# B&R Automation Studio project PLC code - cp (part 24)

```c
		case 8:
			strcpy(txStateDesc, "Waiting homing ");
			TEST_BUSY_CONDITION( !gBlock[1].Status.Motor.xBarsHomed );
			nextState();
			break;

		case 9:

			iTestState = 0;
			TEST_DONE;

			break;

		default:
			break;
	}

}

_TEST test_RemoveTrayMovementMemoryWithKey(void)
{ // Related to https://jira.efi.com/browse/CUBE-963

	if (!gSafetyController.Parameters.xInstalled ){
		iTestState = 0;

		//This 2 lines just for the last TestCase
		strcpy(txTest, "BlockTests Finished!! Congrats!");
		strcpy(txStateDesc, "--");

		TEST_DONE;
	}

	strcpy(txTest, "test_RemoveTrayMovementMemoryWithKey");
	if (strcmp(&txTest, &gSimMachine.Commands.LogTests.Text) != 0){
		strcpy(gSimMachine.Commands.LogTests.Text, txTest); gSimMachine.Commands.LogTests.xCommand = TRUE;
	}
	switch (iTestState)
	{
		case 0:
			gSimMachine.Commands.xToZero = TRUE;
			nextState();
			break;

		case 1:
			strcpy(txStateDesc, "Going to Zero");
			TEST_BUSY_CONDITION( !gMachine.St.Mode.xZero );
			nextState();
			break;

		case 2:
			gSimMachine.Commands.xToAuto = TRUE;
			strcpy(txStateDesc, "Going to Auto");
			TEST_BUSY_CONDITION( !gMachine.St.Mode.xAuto );
			nextState();
			break;

		case 3:
			strcpy(txStateDesc, "Going to Cap");
			TEST_BUSY_CONDITION( gMachine.St.exec.slow < exTimesPreSlow + 3 ); //We'll wait xx scan cycles
			TEST_BUSY_CONDITION( !gMachine.St.Position.xInCap );
			nextState();
			break;

		case 4:
			gSimMachine.Commands.xToZero = TRUE;
			nextState();
			break;

		case 5:
			strcpy(txStateDesc, "Going to Zero");
			TEST_BUSY_CONDITION( !gMachine.St.Mode.xZero );
			nextState();
			break;

		case 6:
			gSimMachine.Commands.xToManual = TRUE;
			strcpy(txStateDesc, "Going to Manual");
			TEST_BUSY_CONDITION( !gMachine.St.Mode.xManual );
			nextState();
			break;

		case 7:
			strcpy(txStateDesc, "Activating the Key");
			TEST_BUSY_CONDITION( gMachine.St.exec.slow < exTimesPreSlow + 2 ); //We'll wait xx scan cycles
			gSimSafetyController.Inputs.xPrinterMaintenanceKey = TRUE;
			nextState();
			break;

		case 8:
			strcpy(txStateDesc, "Send the order to move tray out");
			TEST_BUSY_CONDITION( gMachine.St.exec.slow < exTimesPreSlow + 5 ); //We'll wait xx scan cycles
			gBlock[1].commands.Manual.xManTrayOut = TRUE;
			nextState();
			break;

		case 9:
			strcpy(txStateDesc, "Checking NOT movement");
			TEST_BUSY_CONDITION( gMachine.St.exec.slow < exTimesPreSlow + 20 ); //We'll wait xx scan cycles
			TEST_ASSERT( gBlock[1].In.xTrayIn );
			nextState();
			break;

		case 10:
			strcpy(txStateDesc, "Remove Key");
			TEST_BUSY_CONDITION( gMachine.St.exec.slow < exTimesPreSlow + 5 ); //We'll wait xx scan cycles
			gSimSafetyController.Inputs.xPrinterMaintenanceKey = FALSE;
			nextState();
			break;

		case 11:
			strcpy(txStateDesc, "Checking NOT movement");
			TEST_BUSY_CONDITION( gMachine.St.exec.slow < exTimesPreSlow + 20 ); //We'll wait xx scan cycles
			TEST_ASSERT( gBlock[1].In.xTrayIn );
			nextState();
			break;

		case 12:

			iTestState = 0;

			//This 2 lines just for the last TestCase
			strcpy(txTest, "BlockTests Finished!! Congrats!");
			strcpy(txStateDesc, "--");

			TEST_DONE;
			break;

		default:
			break;
	}

}

/*
B+R UnitTest: This is generated code.
Do not edit! Do not move!
Description: UnitTest Testprogramm infrastructure (TestSet).
LastUpdated: 2024-03-01 15:54:59Z
By B+R UnitTest Helper Version: 2.0.1.59
*/
UNITTEST_FIXTURES(fixtures)
{
	new_TestFixture("test_CleanMachine", test_CleanMachine),
	new_TestFixture("test_GoDownWithTrayError", test_GoDownWithTrayError),
	new_TestFixture("test_GoUpWithTrayError", test_GoUpWithTrayError),
	new_TestFixture("test_GoToPrintInLaboratory", test_GoToPrintInLaboratory),
	new_TestFixture("test_GoToPrintInProduction", test_GoToPrintInProduction),
	new_TestFixture("test_TraySensorErrorWhilePrinting", test_TraySensorErrorWhilePrinting),
	new_TestFixture("test_GoToPrintWhileNSensorsCalibrationAreBeingChecked", test_GoToPrintWhileNSensorsCalibrationAreBeingChecked),
	new_TestFixture("test_ToNotChangeBarsPositionSetpointWhileDetectionSystemMotorIsBeingPositioned", test_ToNotChangeBarsPositionSetpointWhileDetectionSystemMotorIsBeingPositioned),
	new_TestFixture("test_GoToCleanBk1InLaboratory", test_GoToCleanBk1InLaboratory),
	new_TestFixture("test_ReturnToPrintFromClean", test_ReturnToPrintFromClean),
	new_TestFixture("test_RaiseBlocksToCapFromPrinting", test_RaiseBlocksToCapFromPrinting),
	new_TestFixture("test_StopWhenPrint_ReturnPrintingBeforCapPosition", test_StopWhenPrint_ReturnPrintingBeforCapPosition),
	new_TestFixture("test_CriticalAlarmWhilePrinting", test_CriticalAlarmWhilePrinting),
	new_TestFixture("test_GoToMaintenanceWhenInPrintingPositionAndCheckBarsNotMove", test_GoToMaintenanceWhenInPrintingPositionAndCheckBarsNotMove),
	new_TestFixture("test_CuringLedBarJamAlarm", test_CuringLedBarJamAlarm),
	new_TestFixture("test_CameraJamAlarm", test_CameraJamAlarm),
	new_TestFixture("test_TrayBlockMaintenanceKey", test_TrayBlockMaintenanceKey),
	new_TestFixture("test_ToNotExecuteHomingBlockWhileMaintenanceKeyIsActivated", test_ToNotExecuteHomingBlockWhileMaintenanceKeyIsActivated),
	new_TestFixture("test_ToNotExecuteHomingIclaWhileMaintenanceKeyIsActivated", test_ToNotExecuteHomingIclaWhileMaintenanceKeyIsActivated),
	new_TestFixture("test_InkBarJamAlarm", test_InkBarJamAlarm),
	new_TestFixture("test_ToCleanTest", test_ToCleanTest),
	new_TestFixture("test_ToPrintPosTest", test_ToPrintPosTest),
	new_TestFixture("test_InksFailNotEnabledToPrint", test_InksFailNotEnabledToPrint),
	new_TestFixture("test_InksFailEnabledToPrint", test_InksFailEnabledToPrint),
	new_TestFixture("test_NoBentAlarmThcChgOTFly", test_NoBentAlarmThcChgOTFly),
	new_TestFixture("test_NoStopCleanWithNitrLow", test_NoStopCleanWithNitrLow),
	new_TestFixture("test_NoFeederBarsPos", test_NoFeederBarsPos),
	new_TestFixture("test_PneuBlockAls", test_PneuBlockAls),
	new_TestFixture("test_Noz2Jam", test_Noz2Jam),
	new_TestFixture("test_InkTanksAl", test_InkTanksAl),
	new_TestFixture("test_MaintenanceModeInk", test_MaintenanceModeInk),
	new_TestFixture("test_ChillerInksAl", test_ChillerInksAl),
	new_TestFixture("test_NotBlockInAutoIfNotHomed", test_NotBlockInAutoIfNotHomed),
	new_TestFixture("test_RemoveTrayMovementMemoryWithKey", test_RemoveTrayMovementMemoryWithKey),
};

UNITTEST_CALLER_COMPLETE_EXPLICIT(BlockTests, "BlockTests", 0, 0, fixtures, 0, 0, 0);
```

### Program Logical/UnitTest/Tests/CleaningTests

#### CleaningTests.var
```iecst
(********************************************************************
 * COPYRIGHT -- Bernecker + Rainer
 ********************************************************************
 * Program: CleaningTests
 * Author: Jorge Murria
 ********************************************************************
 * Local variables of program CleaningTests
 * General variables - do not change
 ********************************************************************)
(*Describe the test*)
VAR
	Testsuite : UtMgrTestSuite := (Name:='CleaningTests',Description:='Description of the Tests',Type:=utMgrTEST_TYPE_C,MetaInformation:='Some Meta Information can be added here');
END_VAR
(*Variables used in the tests*)
```

#### autoGeneratedFile.c
```c
/*
B+R UnitTest: This is generated code.
Do not edit! Do not move!
Description: UnitTest Testprogramm infrastructure (List of TestSets).
LastUpdated: 2020-05-18 14:29:28Z
By B+R UnitTest Helper Version: 2.0.1.59
*/
#include "UnitTest.h"

UNITTEST_TESTSET_DECLARATION  CleaningTests;

UNITTEST_TESTSET_FIXTURES(utTestSets)
{
	new_TestSet(CleaningTests),
};
UNTITTEST_TESTSET_HANDLER();
```

### Program Logical/UnitTest/Tests/ConsentTests (ANSIC)

#### ConsentTests.var - PVs for the program and test suite
```iecst
(********************************************************************
 * COPYRIGHT -- Bernecker + Rainer
 ********************************************************************
 * Program: ConsentTests
 * Author: Jorge Murria
 ********************************************************************
 * Local variables of program ConsentTests
 * General variables - do not change
 ********************************************************************)
(*Describe the test*)
VAR
	Testsuite : UtMgrTestSuite := (Name:='ConsentTests',Description:='Tests related to the Consents',Type:=utMgrTEST_TYPE_C,MetaInformation:='Some Meta Information can be added here');
END_VAR
(*Variables used in the tests*)
```

#### autoGeneratedFile.c - Auto generated code
```c
/*
B+R UnitTest: This is generated code.
Do not edit! Do not move!
Description: UnitTest Testprogramm infrastructure (List of TestSets).
LastUpdated: 2020-05-18 14:29:28Z
By B+R UnitTest Helper Version: 2.0.1.59
*/
#include "UnitTest.h"

UNITTEST_TESTSET_DECLARATION  ConsentTests;

UNITTEST_TESTSET_FIXTURES(utTestSets)
{
	new_TestSet(ConsentTests),
};
UNTITTEST_TESTSET_HANDLER();
```

### Program Logical/UnitTest/Tests/Cube (ANSIC)

#### Cube.var - PVs for the program and test suite
```iecst
(********************************************************************
 * COPYRIGHT -- Bernecker + Rainer
 ********************************************************************
 * Program: Cube
 * Author: Jorge Murria
 ********************************************************************
 * Local variables of program Cube
 * General variables - do not change
 ********************************************************************)
(*Describe the test*)
VAR
	Testsuite : UtMgrTestSuite := (Name:='Cube',Description:='Description of the Tests',Type:=utMgrTEST_TYPE_C,MetaInformation:='Some Meta Information can be added here');
END_VAR
(*Variables used in the tests*)
```

### Program Logical/UnitTest/Tests/FunctionsTests (ANSIC)

#### FunctionsTests.var - PVs for the program and test suite
```iecst
(********************************************************************
 * COPYRIGHT -- Bernecker + Rainer
 ********************************************************************
 * Program: FunctionsTests
 * Author: Jorge Murria
 ********************************************************************
 * Local variables of program FunctionsTests
 * General variables - do not change
 ********************************************************************)
(*Describe the test*)
VAR
	Testsuite : UtMgrTestSuite := (Name:='FunctionsTests',Description:='Description of the Tests',Type:=utMgrTEST_TYPE_C,MetaInformation:='Some Meta Information can be added here');
END_VAR
(*Variables used in the tests*)
VAR
	TestMediaTracking : ARRAY[0..iMAXTRACKINGARRAY] OF USINT; (*Matrix with the information about if there is Media in the position. Each position corresponds to a cm. Bit 0: L1 , Bit 1 L2*)
	TestBoolMediaTracking : ARRAY[0..iMAXTRACKINGARRAY] OF BOOL; (*Matrix with the information about if there is Media in the position. Each position corresponds to a cm. Bit 0: L1 , Bit 1 L2*)
	xTestMediaDetectionValuesL1 : ARRAY[0..THICK_MAX_UPDATE_VALUES] OF BOOL; (*Matrix with the information about if there is Media in the position. Each position corresponds to a cm. Bit 0: L1 , Bit 1 L2*)
	iIndexArray : UINT;
	TestMediaTrackingInside : ARRAY[0..THICK_MEDIATRACKING_MAX_MEDIA] OF stThicknessCtrl_MediaPosStatus; (*FIFO. Elements enter at the end, and go to First while exiting elements*)
	MediaConfigReseted : stThicknessCtrl_MediaConfig;
	IntensityOutput : ARRAY[0..THICKENERGY_MAX_LAMPS] OF INT;
	EnergyData : stThickCtrl_Energy;
	iIndexProcess : UINT;
	iIndexCross : UINT;
	udResult : UDINT;
	MediaData : stThicknessCtrl_MediaConfig;
	NewMediaStack : ARRAY[0..THICK_MEDIATRACKING_MAX_MEDIA] OF stThicknessCtrl_MediaPosStatus; (*FIFO Stack. Elements enter at the end, and go to First while exiting elements*)
	MediaEnergyRack : ARRAY[0..THICK_MEDIATRACKING_MAX_MEDIA_x2] OF stThickCtrl_Energy; (*Need the memory area for NewMedia and for MediaInside with full data*)
	Stack_iTotalNewMedia : UINT;
	Stack_iTotalNewMediaPos : UINT;
	EnergyRack_iIndex : USINT; (*Index of the next free rack in array*)
	Adresses : ARRAY[0..9] OF UDINT;
END_VAR
```

#### autoGeneratedFile.c - Auto generated code
```c
/*
B+R UnitTest: This is generated code.
Do not edit! Do not move!
Description: UnitTest Testprogramm infrastructure (List of TestSets).
LastUpdated: 2020-05-18 14:29:28Z
By B+R UnitTest Helper Version: 2.0.1.59
*/
#include "UnitTest.h"

UNITTEST_TESTSET_DECLARATION  FunctionsTests;

UNITTEST_TESTSET_FIXTURES(utTestSets)
{
	new_TestSet(FunctionsTests),
};
UNTITTEST_TESTSET_HANDLER();
```

### Program Logical/UnitTest/Tests/LineTests

#### LineTests.var
```iecst
(********************************************************************
 * COPYRIGHT -- Bernecker + Rainer
 ********************************************************************
 * Program: LineTests
 * Author: Jorge Murria
 ********************************************************************
 * Local variables of program LineTests
 * General variables - do not change
 ********************************************************************)
(*Describe the test*)
VAR
	Testsuite : UtMgrTestSuite := (Name:='LineTests',Description:='Description of the Tests',Type:=utMgrTEST_TYPE_C,MetaInformation:='Some Meta Information can be added here');
END_VAR
(*Variables used in the tests*)
```

#### autoGeneratedFile.c
```c
/*
B+R UnitTest: This is generated code.
Do not edit! Do not move!
Description: UnitTest Testprogramm infrastructure (List of TestSets).
LastUpdated: 2020-05-18 14:29:28Z
By B+R UnitTest Helper Version: 2.0.1.59
*/
#include "UnitTest.h"

UNITTEST_TESTSET_DECLARATION  LineTests;

UNITTEST_TESTSET_FIXTURES(utTestSets)
{
	new_TestSet(LineTests),
};
UNTITTEST_TESTSET_HANDLER();
```

#### LineTests.c
```c
/********************************************************************
 * COPYRIGHT -- Bernecker + Rainer
 ********************************************************************
 * Program: ConsentsTests
 * Author: Jorge Murria
 ********************************************************************
 * Prepare machine with basic test to allow proper behabior
 * and starting tasks
 ********************************************************************/

#include <bur/plctypes.h>

#ifdef _DEFAULT_INCLUDES
#include <AsDefault.h>
#endif

#include "UnitTest.h"

#include <stdio.h>
#include <unistd.h>
#include <time.h>         /* clock_t, clock, CLOCKS_PER_SEC */

_LOCAL TIME TimeLast;
_LOCAL TIME endtime;
_LOCAL UDINT diff_t;
_LOCAL STRING stringAux[120];
_LOCAL INT i;
_LOCAL INT iBeltTurns;

#define FALSE 0
#define TRUE 1

void nextState(){
	exTimesPreFast = gMachine.St.exec.fast;
	exTimesPreSlow = gMachine.St.exec.slow;
	iTestState++;
	TimeLast = clock_ms();
	diff_t = diff_t;
	stringAux[120] = stringAux[120];
}

_TEST test_PrintingLine(void)
{
	if (!gMachine.Pt.xControlledByLine ){
		iTestState = 0;
		TEST_DONE;
	}
	strcpy(txTest, "test_PrintingLine");
	switch (iTestState)
	{
		case 0:
			//Line Configuration
			gLine.Inputs.UPSs[1].LoadOnBattery = FALSE;
			gFeeder.Inputs.xModelInput[0]=TRUE;
			gFeeder.ParSw.xEnabled=TRUE;
			gSimMachine.Commands.Media.xMediaIfFeederFeeding = TRUE;
			gPrimer.Inputs.xModelInput[0]=TRUE;
			gPrimer.ParSw.xEnabled=TRUE;
			gPrimer.ParSw.xEnablePriming=TRUE;
			if (gMachine.St.HwData.xIsWater){
				gSarm.Inputs.xModelInput[0]=FALSE;
				gSarm.ParSw.xEnabled=FALSE;
				gDryerAnc.Inputs.xModelInput[0]=TRUE;
				gDryerAnc.ParSw.xEnabled=TRUE;
				gDryerAnc.Inputs.xInRemote=TRUE;
			}
			else {
				gSarm.Inputs.xModelInput[0]=TRUE;
				gSarm.ParSw.xEnabled=TRUE;
				gDryerAnc.Inputs.xModelInput[0]=FALSE;
				gDryerAnc.ParSw.xEnabled=FALSE;
				gDryerAnc.Inputs.xInRemote=FALSE;
			}
			gOverVarnish.Inputs.xModelInput[0]=TRUE;
			gOverVarnish.ParSw.xEnabled=gMachine.St.HwData.xIsWater;
			gOverVarnish.ParSw.xEnablePriming=TRUE;
			gStacker.Inputs.xModelInput[0]=TRUE;
			gStacker.ParSw.xEnabled=TRUE;
			gStacker.Status.Comms.xModuleOk=TRUE;
			gMachine.parSw.Media.rWidth = 1200.0;
			gMachine.parSw.Media.rLength = 1200.0;
			gMachine.parSw.Media.rGap = 100.0;

			gMachine.parSw.Electronics.xRobotReadyL1 = TRUE;
			gSimMachine.Commands.xToZero = TRUE;
			gMachine.parSw.rBeltSpeedSetPoint = 50.0;
			gSimThickCtrl.Commands.xEmptyMediaTracking = TRUE;
			nextState();
			break;

		case 1:
			strcpy(txStateDesc, "Waiting the line to be stopped");
			TEST_BUSY_CONDITION( gMachine.St.exec.fast < exTimesPreFast + 3 );
			TEST_BUSY_CONDITION( !gMachine.St.Mode.xZero );
			TEST_BUSY_CONDITION( gLine.Status != LINE_STOPPED );
			nextState();
			break;

		case 2:
			gSimMachine.Commands.xToAuto = TRUE;
			nextState();
			break;

		case 3:
			strcpy(txStateDesc, "Waiting the machine to be in Auto");
			TEST_BUSY_CONDITION( !gMachine.St.Mode.xAuto );
			gMachine.In.Buttons.xReset = TRUE;
			nextState();
			break;

		case 4:
			strcpy(txStateDesc, "Waiting the machine to be ready");
			TEST_BUSY_CONDITION( gMachine.St.exec.fast < exTimesPreFast + 8 );
			gLine.Commands.Print = TRUE;
			nextState();
			break;

		case 5:
			strcpy(txStateDesc, "Waiting the line to be printing");

			TEST_BUSY_CONDITION( gLine.Status != LINE_PRINTING );
			TEST_ASSERT(gLine.Status == LINE_PRINTING);

			iTestState = 0;
			TEST_DONE;

			break;

		default:
			break;
	}
}

_TEST test_CheckPreprintingPosOrderWithAncillariesEnabled(void)
{
	if (!gMachine.Pt.xControlledByLine ){
		iTestState = 0;
		TEST_DONE;
	}
	strcpy(txTest, "test_CheckPreprintingPosOrderWithAncillariesEnabled");
	switch (iTestState)
	{
		case 0:
			gSimMachine.Commands.xToZero = TRUE;
			nextState();
			break;

		case 1:
			strcpy(txStateDesc, "Waiting the machine to be in Zero");
			TEST_BUSY_CONDITION( gMachine.St.exec.fast < exTimesPreFast + 3 );
			TEST_BUSY_CONDITION( !gMachine.St.Mode.xZero );
			nextState();
			break;

		case 2:
			gSimMachine.Commands.xToAuto = TRUE;
			nextState();
			break;

		case 3:
			strcpy(txStateDesc, "Waiting the machine to be in Auto");
			TEST_BUSY_CONDITION( !gMachine.St.Mode.xAuto );
			gMachine.In.Buttons.xReset = TRUE;
			nextState();
			break;

		case 4:
			strcpy(txStateDesc, "Waiting the machine to be ready");
			TEST_BUSY_CONDITION( gMachine.St.exec.fast < exTimesPreFast + 8 );
			gLine.Commands.Print = TRUE;
			nextState();
			break;

		case 5:
			strcpy(txStateDesc, "Waiting the line to be printing");
			TEST_BUSY_CONDITION( gMachine.St.exec.fast < exTimesPreFast + 8 );
			TEST_BUSY_CONDITION( gLine.Status != LINE_PRINTING );
			nextState();
			break;

		case 6:
			strcpy(txStateDesc, "Waiting the machine to be ready");
			TEST_BUSY_CONDITION( gMachine.St.exec.fast < exTimesPreFast + 8 );
			gLine.Commands.Pause = TRUE;
			nextState();
			break;

		case 7:
			strcpy(txStateDesc, "Waiting the machine to be ready");
			TEST_BUSY_CONDITION( gMachine.St.exec.fast < exTimesPreFast + 8 );
			TEST_BUSY_CONDITION( gLine.Status != LINE_PAUSED );
			TEST_BUSY_CONDITION( !gLine.Orders.Preprinting );
			nextState();
			break;

		case 8:
			strcpy(txStateDesc, "Waiting the line to control stop");
			gLine.Commands.Print = TRUE;
			TEST_BUSY_CONDITION( gLine.Status != LINE_PREPARING_PRINT );
			TEST_ASSERT(gLine.Orders.Preprinting);

			iTestState = 0;
			TEST_DONE;

			break;

		default:
			break;
	}
}

_TEST test_CheckPreprintingPosOrderWithAncillariesDisabled(void)
{
	if (!gMachine.Pt.xControlledByLine ){
		iTestState = 0;
		TEST_DONE;
	}
	strcpy(txTest, "test_CheckPreprintingPosOrderWithAncillariesDisabled");
	switch (iTestState)
	{
		case 0:
			gSimMachine.Commands.xToZero = TRUE;
			gFeeder.ParSw.xEnabled=FALSE;
			gPrimer.ParSw.xEnabled=FALSE;
			gSarm.ParSw.xEnabled=FALSE;
			nextState();
			break;

		case 1:
			strcpy(txStateDesc, "Waiting the machine to be in Zero");
			TEST_BUSY_CONDITION( gMachine.St.exec.fast < exTimesPreFast + 3 );
			TEST_BUSY_CONDITION( !gMachine.St.Mode.xZero );
			nextState();
			break;

		case 2:
			gSimMachine.Commands.xToAuto = TRUE;
			nextState();
			break;

		case 3:
			strcpy(txStateDesc, "Waiting the machine to be in Auto");
			TEST_BUSY_CONDITION( !gMachine.St.Mode.xAuto );
			gMachine.In.Buttons.xReset = TRUE;
			nextState();
			break;

		case 4:
			strcpy(txStateDesc, "Waiting the machine to be ready");
			TEST_BUSY_CONDITION( gMachine.St.exec.fast < exTimesPreFast + 8 );
			gLine.Commands.Print = TRUE;
			nextState();
			break;

		case 5:
			strcpy(txStateDesc, "Waiting the line to be printing");
			TEST_BUSY_CONDITION( gMachine.St.exec.fast < exTimesPreFast + 8 );
			TEST_BUSY_CONDITION( gLine.Status != LINE_PRINTING );
			nextState();
			break;

		case 6:
			strcpy(txStateDesc, "Waiting the machine to be ready");
			TEST_BUSY_CONDITION( gMachine.St.exec.fast < exTimesPreFast + 8 );
			gLine.Commands.Pause = TRUE;
			nextState();
			break;

		case 7:
			strcpy(txStateDesc, "Waiting the machine to be ready");
			TEST_BUSY_CONDITION( gMachine.St.exec.fast < exTimesPreFast + 8 );
			TEST_BUSY_CONDITION( gLine.Status != LINE_PAUSED );
			nextState();
			break;

		case 8:
			strcpy(txStateDesc, "Waiting the line to control stop");
			gLine.Commands.Print = TRUE;
			TEST_BUSY_CONDITION( gLine.Status != LINE_PRINTING );
			TEST_ASSERT(!gLine.Orders.Preprinting);

			gFeeder.ParSw.xEnabled=TRUE;
			gPrimer.ParSw.xEnabled=TRUE;
			gSarm.ParSw.xEnabled=TRUE;

			iTestState = 0;
			TEST_DONE;

			break;

		default:
			break;
	}
}

_TEST test_EmptyingBeltLine(void)
{
	if (!gMachine.Pt.xControlledByLine ){
		iTestState = 0;
		TEST_DONE;
	}
	strcpy(txTest, "test_EmptyingBeltLine");
	switch (iTestState)
	{
		case 0:
			gSimMachine.Commands.xToZero = TRUE;
			nextState();
			break;

		case 1:
			strcpy(txStateDesc, "Waiting the machine to be in Zero");
			TEST_BUSY_CONDITION( gMachine.St.exec.fast < exTimesPreFast + 3 );
			TEST_BUSY_CONDITION( !gMachine.St.Mode.xZero );
			TEST_BUSY_CONDITION( gLine.Status != LINE_STOPPED );
			nextState();
			break;

		case 2:
			gSimMachine.Commands.xToAuto = TRUE;
			nextState();
			break;

		case 3:
			strcpy(txStateDesc, "Waiting the machine to be in Auto");
			TEST_BUSY_CONDITION( !gMachine.St.Mode.xAuto );
			gMachine.In.Buttons.xReset = TRUE;
			nextState();
			break;

		case 4:
			strcpy(txStateDesc, "Waiting the machine to be ready");
			TEST_BUSY_CONDITION( gMachine.St.exec.fast < exTimesPreFast + 8 );
			gLine.Commands.EmptyBelt = TRUE;
			nextState();
			break;

		case 5:
			strcpy(txStateDesc, "Waiting the line to be emptying belts");

			TEST_BUSY_CONDITION( gLine.Status != LINE_BELT_EMPTYING );
			TEST_ASSERT(gLine.Status == LINE_BELT_EMPTYING);
			TEST_ASSERT(!gThicknessCtrl.Outputs.xEnableMediaSignalToCb);
			gLine.Commands.Stop = TRUE;
			nextState();
			break;

		case 6:
			strcpy(txStateDesc, "Waiting the machine to be empty");
			TEST_BUSY_CONDITION( gLine.Status==LINE_IDLE );

			iTestState = 0;
			TEST_DONE;

			break;

		default:
			break;
	}
}

/* --- Test for DELOREAN-955 Check not curing when bars in cap position --- */
_TEST test_EmptyingBeltLineWithMediaEntering(void)
{
	if (!gMachine.Pt.xControlledByLine ){
		iTestState = 0;
		TEST_DONE;
	}
	strcpy(txTest, "test_EmptyingBeltLineWithMediaEntering");
	//If the Test makes non sense, not execute it. Only check for color cure because the behaviour is the same for all
	if (!gCuringLed[iIndexColorCuringLedBar].Parameters.xInstalled ){
		iTestState = 0;
		TEST_DONE;
	}

	switch (iTestState)
	{
		case 0:
			gSimMachine.Commands.xToZero = TRUE;
			nextState();
			break;

		case 1:
			strcpy(txStateDesc, "Waiting the machine to be in Zero");
			TEST_BUSY_CONDITION( gMachine.St.exec.fast < exTimesPreFast + 3 );
			TEST_BUSY_CONDITION( !gMachine.St.Mode.xZero );
			TEST_BUSY_CONDITION( gLine.Status != LINE_STOPPED );
			nextState();
			break;

		case 2:
			gSimMachine.Commands.xToAuto = TRUE;
			nextState();
			break;

		case 3:
			strcpy(txStateDesc, "Waiting the machine to be in Auto");
			TEST_BUSY_CONDITION( !gMachine.St.Mode.xAuto );
			gMachine.In.Buttons.xReset = TRUE;
			nextState();
			break;

		case 4:
			strcpy(txStateDesc, "Waiting the machine to be ready");
			TEST_BUSY_CONDITION( gMachine.St.exec.fast < exTimesPreFast + 8 );
			gSimMachine.Commands.Media.xContinuousMediaPresent = TRUE;
			gLine.Commands.EmptyBelt = TRUE;
			nextState();
			break;

		case 5:
			strcpy(txStateDesc, "Waiting the line to be emptying belts");
			TEST_BUSY_CONDITION( gLine.Status != LINE_BELT_EMPTYING );
			TEST_ASSERT(gLine.Status == LINE_BELT_EMPTYING);
			TEST_ASSERT(!gThicknessCtrl.Outputs.xEnableMediaSignalToCb);
			/*gSimMachine.Commands.Media.xContinuousMediaPresent = TRUE;*/
			nextState();
			break;

		case 6:
			strcpy(txStateDesc, "Check that curing leds are not curing media");
			TEST_BUSY_CONDITION(!gThicknessCtrl.status.MediaPosition.L1.Color.xMediaInLedPosition);
			if(gMachine.St.Position.xInCap){
				TEST_ASSERT(!gCuringLed[iIndexColorCuringLedBar].Commands.RunCuring && gMachine.St.Position.xInCap);
			}
			gSimMachine.Commands.Media.xContinuousMediaPresent = FALSE;
			gLine.Commands.EmptyBelt = FALSE;
			iTestState = 0;
			TEST_DONE;

			break;

		default:
			break;
	}
}
	/* --- End Test for DELOREAN-955 --- */

_TEST test_CleaningLine(void)
{
	if (!gMachine.Pt.xControlledByLine ){
		iTestState = 0;
		TEST_DONE;
	}
	strcpy(txTest, "test_CleaningLine");
	switch (iTestState)
	{
		case 0:
			gSimMachine.Commands.xToZero = TRUE;
			nextState();
			break;

		case 1:
			strcpy(txStateDesc, "Waiting the machine to be in Zero");
			TEST_BUSY_CONDITION( gMachine.St.exec.fast < exTimesPreFast + 3 );
			TEST_BUSY_CONDITION( !gMachine.St.Mode.xZero );
			TEST_BUSY_CONDITION( gLine.Status != LINE_STOPPED );
			nextState();
			break;

		case 2:
			gSimMachine.Commands.xToAuto = TRUE;
			nextState();
			break;

		case 3:
			strcpy(txStateDesc, "Waiting the machine to be in Auto");
			TEST_BUSY_CONDITION( !gMachine.St.Mode.xAuto );
			gMachine.In.Buttons.xReset = TRUE;
			nextState();
			break;

		case 4:
			strcpy(txStateDesc, "Waiting the machine to be ready");
			TEST_BUSY_CONDITION( gMachine.St.exec.fast < exTimesPreFast + 8 );
			gLine.Commands.Clean = TRUE;
			nextState();
			break;

		case 5:
			strcpy(txStateDesc, "Waiting the line to be cleaning");

			TEST_BUSY_CONDITION( gLine.Status != LINE_CLEANINGPH );
			TEST_ASSERT(gLine.Status == LINE_CLEANINGPH);

			iTestState = 0;
			TEST_DONE;

			break;

		default:
			break;
	}
}

_TEST test_PoweringOffLine(void)
{
	if (!gMachine.Pt.xControlledByLine ){
		iTestState = 0;
		TEST_DONE;
	}
	strcpy(txTest, "test_PoweringOffLine");
	switch (iTestState)
	{
		case 0:
			gSimMachine.Commands.xToZero = TRUE;
			nextState();
			break;

		case 1:
			strcpy(txStateDesc, "Waiting the machine to be in Zero");
			TEST_BUSY_CONDITION( gMachine.St.exec.fast < exTimesPreFast + 3 );
			TEST_BUSY_CONDITION( !gMachine.St.Mode.xZero );
			TEST_BUSY_CONDITION( gLine.Status != LINE_STOPPED );
			nextState();
			break;

		case 2:
			gSimMachine.Commands.xToAuto = TRUE;
			nextState();
			break;

		case 3:
			strcpy(txStateDesc, "Waiting the machine to be in Auto");
			TEST_BUSY_CONDITION( !gMachine.St.Mode.xAuto );
			gMachine.In.Buttons.xReset = TRUE;
			nextState();
			break;

		case 4:
			strcpy(txStateDesc, "Waiting the machine to be ready");
			TEST_BUSY_CONDITION( gMachine.St.exec.fast < exTimesPreFast + 8 );
			gLine.OrdersSw.Shutdown = TRUE;
			nextState();
			break;

		case 5:
			strcpy(txStateDesc, "Waiting the line to power off all devices");
			TEST_BUSY_CONDITION( gLine.Status != LINE_POWERING_OFF );
			TEST_ASSERT(gLine.Status == LINE_POWERING_OFF);
			nextState();
			break;

		case 6:
			strcpy(txStateDesc, "Waiting the machine to be not powered");
			TEST_BUSY_CONDITION( gLine.Status != LINE_NOT_POWERED );
			TEST_ASSERT(gLine.Status == LINE_NOT_POWERED);
			gLine.OrdersSw.Shutdown = FALSE;
			nextState();
			break;

		case 7:
			strcpy(txStateDesc, "Waiting the machine to be ready");
			TEST_BUSY_CONDITION( gLine.Status != LINE_STOPPED );
			TEST_ASSERT(gLine.Status == LINE_STOPPED);

			iTestState = 0;
			TEST_DONE;

			break;

		default:
			break;
	}
}

_TEST test_CleaningByTilesLine(void)
{
	if (!gMachine.Pt.xControlledByLine ){
		iTestState = 0;
		TEST_DONE;
	}
	strcpy(txTest, "test_CleaningByTilesLine");
	switch (iTestState)
	{
		case 0:
			gSimMachine.Commands.xToZero = TRUE;
			gMachine.parSw.Clean.xCleanSystemByPieces = FALSE;
			gMachine.parSw.Clean.iPiecesNumberToCleanL1 = 10;
			nextState();
			break;

		case 1:
			strcpy(txStateDesc, "Waiting the machine to be in Zero");
			TEST_BUSY_CONDITION( gMachine.St.exec.fast < exTimesPreFast + 3 );
			TEST_BUSY_CONDITION( !gMachine.St.Mode.xZero );
			gSimThickCtrl.Commands.xEmptyMediaTracking = TRUE;
			TEST_BUSY_CONDITION( gLine.Status != LINE_STOPPED );
			nextState();
			break;

		case 2:
			gSimMachine.Commands.xToAuto = TRUE;
			nextState();
			break;

		case 3:
			strcpy(txStateDesc, "Waiting the machine to be in Auto");
			TEST_BUSY_CONDITION( !gMachine.St.Mode.xAuto );
			gMachine.In.Buttons.xReset = TRUE;
			nextState();
			break;

		case 4:
			strcpy(txStateDesc, "Waiting the machine to be ready");
			TEST_BUSY_CONDITION( gMachine.St.exec.fast < exTimesPreFast + 8 );
			gLine.Commands.Print = TRUE;
			nextState();
			break;

		case 5:
			strcpy(txStateDesc, "Waiting the line to be printing");
			TEST_BUSY_CONDITION( gLine.Status != LINE_PRINTING );
			gMachine.parSw.Clean.xCleanSystemByPieces = TRUE;
			gSimMachine.Commands.Media.xContinuousMediaPresent = TRUE;
			nextState();
			break;

		case 6:
			strcpy(txStateDesc, "Waiting the line to be pausing");
			TEST_BUSY_CONDITION( gLine.Status != LINE_PAUSING );
			gSimMachine.Commands.Media.xContinuousMediaPresent = FALSE;
			nextState();
			break;

		case 7:
			strcpy(txStateDesc, "Waiting the line to be cleaning");
			TEST_BUSY_CONDITION( !gLine.StatusSummary.xCleaning );
			TEST_ASSERT(gThicknessCtrl.status.Belt.xBeltEmpty );
			gMachine.parSw.Clean.xCleanSystemByPieces = FALSE;
			nextState();
			break;

		case 8:
			strcpy(txStateDesc, "Waiting the line to be cleaning");
			TEST_BUSY_CONDITION( gLine.Status != LINE_CLEANINGPH );
			nextState();
			break;

		case 9:
			strcpy(txStateDesc, "Waiting the line to be printing");
			TEST_BUSY_CONDITION( gLine.Status != LINE_PRINTING );
			TEST_ASSERT(gBelt.states.xRuningBelt);
			TEST_ASSERT(gLine.Status == LINE_PRINTING);

			iTestState = 0;
			TEST_DONE;

			break;

		default:
			break;
	}
}

_TEST test_ReturnToPrintFromCleanLine(void)
{
	if (!gMachine.Pt.xControlledByLine ){
		iTestState = 0;
		TEST_DONE;
	}
	strcpy(txTest, "test_ReturnToPrintFromCleanLine");
	switch (iTestState)
	{
		case 0:
			gSimMachine.Commands.xToZero = TRUE;
			nextState();
			break;

		case 1:
			strcpy(txStateDesc, "Waiting the machine to be in Zero");
			TEST_BUSY_CONDITION( gMachine.St.exec.fast < exTimesPreFast + 3 );
			TEST_BUSY_CONDITION( !gMachine.St.Mode.xZero );
			nextState();
			break;

		case 2:
			gSimMachine.Commands.xToAuto = TRUE;
			nextState();
			break;

		case 3:
			strcpy(txStateDesc, "Waiting the machine to be in Auto");
			TEST_BUSY_CONDITION( !gMachine.St.Mode.xAuto );
			gMachine.In.Buttons.xReset = TRUE;
			nextState();
			break;

		case 4:
			strcpy(txStateDesc, "Waiting the machine to be ready");
			TEST_BUSY_CONDITION( gMachine.St.exec.fast < exTimesPreFast + 8 );
			gLine.Commands.Print = TRUE;
			nextState();
			break;

		case 5:
			strcpy(txStateDesc, "Waiting the line to be printing");
			TEST_BUSY_CONDITION( gLine.Status != LINE_PRINTING );
			nextState();
			break;

		case 6:
			strcpy(txStateDesc, "Waiting the machine to be ready");
			TEST_BUSY_CONDITION( gMachine.St.exec.fast < exTimesPreFast + 8 );
			gLine.Commands.Clean = TRUE;
			TEST_BUSY_CONDITION( gLine.Status != LINE_PAUSED );
			nextState();
			break;

		case 7:
			strcpy(txStateDesc, "Waiting the line to be cleaning");
			TEST_BUSY_CONDITION( gMachine.St.exec.fast < exTimesPreFast + 8 );
			TEST_BUSY_CONDITION( gLine.Status != LINE_CLEANED );
			nextState();
			break;

		case 8:
			strcpy(txStateDesc, "Waiting the line to return printing");
			TEST_BUSY_CONDITION( gMachine.St.exec.fast < exTimesPreFast + 8 );
			TEST_BUSY_CONDITION( gLine.Status == LINE_PREPARING_PRINT || gLine.Status == LINE_STARTING_PRINTING );
			TEST_ASSERT(gLine.Status == LINE_PRINTING);

			iTestState = 0;
			TEST_DONE;

			break;

		default:
			break;
	}
}

_TEST test_ReturnToPrintFromPauseLine(void)
{
	if (!gMachine.Pt.xControlledByLine ){
		iTestState = 0;
		TEST_DONE;
	}
	strcpy(txTest, "test_ReturnToPrintFromPauseLine");
	switch (iTestState)
	{
		case 0:
			gSimMachine.Commands.xToZero = TRUE;
			nextState();
			break;

		case 1:
			strcpy(txStateDesc, "Waiting the machine to be in Zero");
			TEST_BUSY_CONDITION( gMachine.St.exec.fast < exTimesPreFast + 3 );
			TEST_BUSY_CONDITION( !gMachine.St.Mode.xZero );
			nextState();
			break;

		case 2:
			gSimMachine.Commands.xToAuto = TRUE;
			nextState();
			break;

		case 3:
			strcpy(txStateDesc, "Waiting the machine to be in Auto");
			TEST_BUSY_CONDITION( !gMachine.St.Mode.xAuto );
			gMachine.In.Buttons.xReset = TRUE;
			nextState();
			break;

		case 4:
			strcpy(txStateDesc, "Waiting the machine to be ready");
			TEST_BUSY_CONDITION( gMachine.St.exec.fast < exTimesPreFast + 8 );
			gLine.Commands.Print = TRUE;
			nextState();
			break;

		case 5:
			strcpy(txStateDesc, "Waiting the line to be printing");
			TEST_BUSY_CONDITION( gMachine.St.exec.fast < exTimesPreFast + 8 );
			TEST_BUSY_CONDITION( gLine.Status != LINE_PRINTING );
			nextState();
			break;

		case 6:
			strcpy(txStateDesc, "Waiting the machine to be ready");
			TEST_BUSY_CONDITION( gMachine.St.exec.fast < exTimesPreFast + 8 );
			gMachine.In.Buttons.xStart = TRUE;
			nextState();
			break;

		case 7:
			strcpy(txStateDesc, "Waiting the line to pause");
			TEST_BUSY_CONDITION( gLine.Status != LINE_PAUSED );
			gMachine.In.Buttons.xStart = FALSE;
			gLine.Commands.Print = TRUE;
			nextState();
			break;

		case 8:
			strcpy(txStateDesc, "Waiting the line to return printing");
			TEST_BUSY_CONDITION( gMachine.St.exec.fast < exTimesPreFast + 8 );
			TEST_BUSY_CONDITION( gLine.Status == LINE_PREPARING_PRINT || gLine.Status == LINE_STARTING_PRINTING );
			TEST_ASSERT(gLine.Status == LINE_PRINTING);

			iTestState = 0;
			TEST_DONE;

			break;

		default:
			break;
	}
}

_TEST test_ReturnToPauseFromCleanedLine(void)
{
	if (!gMachine.Pt.xControlledByLine ){
		iTestState = 0;
		TEST_DONE;
	}
	strcpy(txTest, "test_ReturnToPauseFromCleanedLine");
	switch (iTestState)
	{
		case 0:
			gSimMachine.Commands.xToZero = TRUE;
			nextState();
			break;

		case 1:
			strcpy(txStateDesc, "Waiting the machine to be in Zero");
			TEST_BUSY_CONDITION( gMachine.St.exec.fast < exTimesPreFast + 3 );
			TEST_BUSY_CONDITION( !gMachine.St.Mode.xZero );
			nextState();
			break;

		case 2:
			gSimMachine.Commands.xToAuto = TRUE;
			nextState();
			break;

		case 3:
			strcpy(txStateDesc, "Waiting the machine to be in Auto");
			TEST_BUSY_CONDITION( !gMachine.St.Mode.xAuto );
			gMachine.In.Buttons.xReset = TRUE;
			nextState();
			break;

		case 4:
			strcpy(txStateDesc, "Waiting the machine to be ready");
			TEST_BUSY_CONDITION( gMachine.St.exec.fast < exTimesPreFast + 8 );
			gLine.Commands.Print = TRUE;
			nextState();
			break;

		case 5:
			strcpy(txStateDesc, "Waiting the line to be printing");
			TEST_BUSY_CONDITION( gMachine.St.exec.fast < exTimesPreFast + 8 );
			TEST_BUSY_CONDITION( gLine.Status != LINE_PRINTING );
			nextState();
			break;

		case 6:
			strcpy(txStateDesc, "Waiting the machine to be ready");
			TEST_BUSY_CONDITION( gMachine.St.exec.fast < exTimesPreFast + 8 );
			gMachine.In.Buttons.xStart = TRUE; //Entering pause using phyisical start button
			nextState();
			break;

		case 7:
			strcpy(txStateDesc, "Waiting the line to pause");
			TEST_BUSY_CONDITION( gLine.Status != LINE_PAUSED );
			gMachine.In.Buttons.xStart = FALSE;
			gLine.Commands.Clean = TRUE;
			nextState();
			break;

		case 8:
			strcpy(txStateDesc, "Waiting the line to be cleaning");
			TEST_BUSY_CONDITION( gMachine.St.exec.fast < exTimesPreFast + 8 );
			TEST_BUSY_CONDITION( !gLine.StatusSummary.xCleaning );
			nextState();
			break;

		case 9:
			strcpy(txStateDesc, "Waiting the line to finish cleaning");
			TEST_BUSY_CONDITION( gMachine.St.exec.fast < exTimesPreFast + 8 );
			TEST_BUSY_CONDITION( gLine.StatusSummary.xCleaning );
			nextState();
			break;

		case 10:
			strcpy(txStateDesc, "Waiting the line to return pausing");
			TEST_BUSY_CONDITION( gLine.Status == LINE_PAUSING );
			nextState();
			break;

		case 11:
			strcpy(txStateDesc, "Waiting the line to be paused");
			TEST_BUSY_CONDITION( !gLine.Status == LINE_PAUSED );
			TEST_ASSERT(gLine.Status == LINE_PAUSED);

			iTestState = 0;
			TEST_DONE;

			break;

		default:
			break;
	}
}

_TEST test_ControlStopWhilePrintingLine(void)
{
	if (!gMachine.Pt.xControlledByLine ){
		iTestState = 0;
		TEST_DONE;
	}
	strcpy(txTest, "test_ControlStopWhilePrintingLine");
	switch (iTestState)
	{
		case 0:
			gSimMachine.Commands.xToZero = TRUE;
			nextState();
			break;

		case 1:
			strcpy(txStateDesc, "Waiting the machine to be in Zero");
			TEST_BUSY_CONDITION( gMachine.St.exec.fast < exTimesPreFast + 3 );
			TEST_BUSY_CONDITION( !gMachine.St.Mode.xZero );
			nextState();
			break;

		case 2:
			gSimMachine.Commands.xToAuto = TRUE;
			nextState();
			break;

		case 3:
			strcpy(txStateDesc, "Waiting the machine to be in Auto");
			TEST_BUSY_CONDITION( !gMachine.St.Mode.xAuto );
			gMachine.In.Buttons.xReset = TRUE;
			nextState();
			break;

		case 4:
			strcpy(txStateDesc, "Waiting the machine to be ready");
			TEST_BUSY_CONDITION( gMachine.St.exec.fast < exTimesPreFast + 8 );
			gLine.Commands.Print = TRUE;
			nextState();
			break;

		case 5:
			strcpy(txStateDesc, "Waiting the line to be printing");
			TEST_BUSY_CONDITION( gMachine.St.exec.fast < exTimesPreFast + 8 );
			TEST_BUSY_CONDITION( gLine.Status != LINE_PRINTING );
			if (gEdgeHoldDown.parSw.xEnable ){
				TEST_ASSERT(gEdgeHoldDown.status.xAdjustedToMedia);
				TEST_ASSERT(!gEdgeHoldDown.parameters.xEnableMovements);
			}
			TEST_ASSERT(gTransVacuum[1].Parameters.rVacPressureSetPointPerc == gTransVacuum[1].parSw.rVacPressureSetPointPerc);
			rPreviousVacPressureSp = gTransVacuum[1].Parameters.rVacPressureSetPointPerc;
			nextState();
			break;

		case 6:
			strcpy(txStateDesc, "Waiting the line to control stop");
			gLine.Commands.Stop = TRUE;
			TEST_BUSY_CONDITION( gLine.Status != LINE_CONTROLLED_STOP );
			TEST_ASSERT(gTransVacuum[1].Parameters.rVacPressureSetPointPerc == rPreviousVacPressureSp);
			nextState();
			break;

		case 7:
			strcpy(txStateDesc, "Waiting the line to be stopped");
			gMachine.In.Buttons.xReset = TRUE;
			TEST_BUSY_CONDITION( gLine.Status == LINE_CONTROLLED_STOP );
			TEST_ASSERT(gLine.Status == LINE_STOPPED);
			if (gEdgeHoldDown.parSw.xEnable ){
				TEST_ASSERT(gEdgeHoldDown.status.iSystemState==EHD_IDLE);
				TEST_ASSERT(gPairedMotors[1].Motor[1].Inputs.xMinPositionReached);
				TEST_ASSERT(gPairedMotors[1].Motor[2].Inputs.xMinPositionReached);
				TEST_ASSERT(gPairedMotors[2].Motor[1].Inputs.xMaxPositionReached);
				TEST_ASSERT(gPairedMotors[2].Motor[2].Inputs.xMaxPositionReached);
			}

			iTestState = 0;
			TEST_DONE;

			break;

		default:
			break;
	}
}

_TEST test_ControlStopDueToSwCriticalConditionWhilePrintingLine(void)
{
	if (!gMachine.Pt.xControlledByLine ){
		iTestState = 0;
		TEST_DONE;
	}
	strcpy(txTest, "test_ControlStopDueToSwCriticalConditionWhilePrintingLine");
	switch (iTestState)
	{
		case 0:
			gSimMachine.Commands.xToZero = TRUE;
			nextState();
			break;

		case 1:
			strcpy(txStateDesc, "Waiting the machine to be in Zero");
			TEST_BUSY_CONDITION( gMachine.St.exec.fast < exTimesPreFast + 3 );
			TEST_BUSY_CONDITION( !gMachine.St.Mode.xZero );
			nextState();
			break;

		case 2:
			gSimMachine.Commands.xToAuto = TRUE;
			nextState();
			break;

		case 3:
			strcpy(txStateDesc, "Waiting the machine to be in Auto");
			TEST_BUSY_CONDITION( !gMachine.St.Mode.xAuto );
			gMachine.In.Buttons.xReset = TRUE;
			nextState();
			break;

		case 4:
			strcpy(txStateDesc, "Waiting the machine to be ready");
			TEST_BUSY_CONDITION( gMachine.St.exec.fast < exTimesPreFast + 8 );
			gLine.Commands.Print = TRUE;
			nextState();
			break;

		case 5:
			strcpy(txStateDesc, "Waiting the line to be printing");
			TEST_BUSY_CONDITION( gMachine.St.exec.fast < exTimesPreFast + 8 );
			TEST_BUSY_CONDITION( gLine.Status != LINE_PRINTING );
			nextState();
			break;

		case 6:
			strcpy(txStateDesc, "Waiting the line to control stop");
			gMachine.parSw.UI.xCriticalCondition = TRUE;
			TEST_BUSY_CONDITION( gLine.Status != LINE_CONTROLLED_STOP );
			gMachine.parSw.UI.xCriticalCondition = FALSE;
			nextState();
			break;

		case 7:
			strcpy(txStateDesc, "Waiting the line to be stopped");
			gMachine.In.Buttons.xReset = TRUE;
			TEST_BUSY_CONDITION( gLine.Status == LINE_CONTROLLED_STOP );
			TEST_ASSERT(gLine.Status == LINE_STOPPED);

			iTestState = 0;
			TEST_DONE;

			break;

		default:
			break;
	}
}

_TEST test_PauseDueToFeederErrorWhilePrintingLine(void)
{
	if (!gMachine.Pt.xControlledByLine ){
		iTestState = 0;
		TEST_DONE;
	}
	strcpy(txTest, "test_PauseDueToFeederErrorWhilePrintingLine");
	switch (iTestState)
	{
		case 0:
			gSimMachine.Commands.xToZero = TRUE;
			nextState();
			break;

		case 1:
			strcpy(txStateDesc, "Waiting the machine to be in Zero");
			TEST_BUSY_CONDITION( gMachine.St.exec.fast < exTimesPreFast + 3 );
			TEST_BUSY_CONDITION( !gMachine.St.Mode.xZero );
			nextState();
			break;

		case 2:
			gSimMachine.Commands.xToAuto = TRUE;
			nextState();
			break;

		case 3:
			strcpy(txStateDesc, "Waiting the machine to be in Auto");
			TEST_BUSY_CONDITION( !gMachine.St.Mode.xAuto );
			gMachine.In.Buttons.xReset = TRUE;
			nextState();
			break;

		case 4:
			strcpy(txStateDesc, "Waiting the machine to be ready");
			TEST_BUSY_CONDITION( gMachine.St.exec.fast < exTimesPreFast + 8 );
			gLine.Commands.Print = TRUE;
			nextState();
			break;

		case 5:
			strcpy(txStateDesc, "Waiting the line to be printing");
			TEST_BUSY_CONDITION( gMachine.St.exec.fast < exTimesPreFast + 8 );
			TEST_BUSY_CONDITION( gLine.Status != LINE_PRINTING );
			nextState();
			break;

		case 6:
			strcpy(txStateDesc, "Waiting the line to pause");
			gSimFeeder.Commands.CreateError = TRUE;
			TEST_BUSY_CONDITION( gLine.Status != LINE_PAUSING );
			gSimFeeder.Commands.CreateError = FALSE;
			nextState();
			break;

		case 7:
			strcpy(txStateDesc, "Waiting the line to be paused");
			TEST_BUSY_CONDITION( gMachine.St.exec.fast < exTimesPreFast + 8 );
			TEST_BUSY_CONDITION( gLine.Status == LINE_PAUSING );
			TEST_ASSERT(gLine.Status == LINE_PAUSED);
			TEST_ASSERT(gFeeder.Alarms.xCriticalAlarm);
			nextState();
			break;

		case 8:
			strcpy(txStateDesc, "Sending to print");
			gLine.Commands.Print = TRUE;
			TEST_BUSY_CONDITION( gFeeder.Alarms.xCriticalAlarm );
			TEST_ASSERT(!gFeeder.Alarms.xCriticalAlarm);
			TEST_ASSERT(gLine.Status == LINE_PREPARING_PRINT);

			iTestState = 0;
			TEST_DONE;

			break;

		default:
			break;
	}
}

_TEST test_GoingToPauseWhenPrintCommandIsReceivedWhileFeederIsInErrorLine(void)
{
	if (!gMachine.Pt.xControlledByLine ){
		iTestState = 0;
		TEST_DONE;
	}
	strcpy(txTest, "test_GoingToPauseWhenPrintCommandIsReceivedWhileFeederIsInErrorLine");
	switch (iTestState)
	{
		case 0:
			gSimMachine.Commands.xToZero = TRUE;
			nextState();
			break;

		case 1:
			strcpy(txStateDesc, "Waiting the machine to be in Zero");
			TEST_BUSY_CONDITION( gMachine.St.exec.fast < exTimesPreFast + 3 );
			TEST_BUSY_CONDITION( !gMachine.St.Mode.xZero );
			nextState();
			break;

		case 2:
			gSimMachine.Commands.xToAuto = TRUE;
			nextState();
			break;

		case 3:
			strcpy(txStateDesc, "Waiting the machine to be in Auto");
			TEST_BUSY_CONDITION( !gMachine.St.Mode.xAuto );
			gMachine.In.Buttons.xReset = TRUE;
			nextState();
			break;

		case 4:
			strcpy(txStateDesc, "Waiting the machine to be ready");
			TEST_BUSY_CONDITION( gMachine.St.exec.fast < exTimesPreFast + 8 );
			gLine.Commands.Print = TRUE;
			nextState();
			break;

		case 5:
			strcpy(txStateDesc, "Waiting the line to be printing");
			TEST_BUSY_CONDITION( gMachine.St.exec.fast < exTimesPreFast + 8 );
			TEST_BUSY_CONDITION( gLine.Status != LINE_PRINTING );
			nextState();
			break;

		case 6:
			strcpy(txStateDesc, "Waiting the line to pause");
			gSimFeeder.Commands.CreateError = TRUE;
			TEST_BUSY_CONDITION( gLine.Status != LINE_PAUSING );
			nextState();
			break;

		case 7:
			strcpy(txStateDesc, "Waiting the line to be paused");
			TEST_BUSY_CONDITION( gMachine.St.exec.fast < exTimesPreFast + 8 );
			TEST_BUSY_CONDITION( gLine.Status == LINE_PAUSING );
			TEST_ASSERT(gLine.Status == LINE_PAUSED);
			nextState();
			break;

		case 8:
			strcpy(txStateDesc, "Sending to print");
			gLine.Commands.Print = TRUE;
			TEST_BUSY_CONDITION(gLine.Status == LINE_PAUSED);
			TEST_ASSERT(gLine.StatusSummary.xPrinting);
			nextState();
			break;

		case 9:
			strcpy(txStateDesc, "Waiting the line to be paused again");
			TEST_BUSY_CONDITION(gLine.StatusSummary.xPrinting);
			TEST_ASSERT(gLine.StatusSummary.xPausing);
			TEST_ASSERT(gFeeder.Alarms.xCriticalAlarm);
			gSimFeeder.Commands.CreateError = FALSE;

			iTestState = 0;
			TEST_DONE;

			break;

		default:
			break;
	}
}

_TEST test_ControlStopWhilePrepareToPrintLine(void)
{
	if (!gMachine.Pt.xControlledByLine ){
		iTestState = 0;
		TEST_DONE;
	}
	strcpy(txTest, "test_ControlStopWhilePrepareToPrintLine");
	switch (iTestState)
	{
		case 0:
			gSimMachine.Commands.xToZero = TRUE;
			nextState();
			break;

		case 1:
			strcpy(txStateDesc, "Waiting the machine to be in Zero");
			TEST_BUSY_CONDITION( gMachine.St.exec.fast < exTimesPreFast + 3 );
			TEST_BUSY_CONDITION( !gMachine.St.Mode.xZero );
			nextState();
			break;

		case 2:
			gSimMachine.Commands.xToAuto = TRUE;
			nextState();
			break;

		case 3:
			strcpy(txStateDesc, "Waiting the machine to be in Auto");
			TEST_BUSY_CONDITION( gMachine.St.exec.fast < exTimesPreFast + 8 );
			TEST_BUSY_CONDITION( !gMachine.St.Mode.xAuto );
			gMachine.In.Buttons.xReset = TRUE;
			nextState();
			break;

		case 4:
			strcpy(txStateDesc, "Waiting the machine to be ready");
			TEST_BUSY_CONDITION( gMachine.St.exec.fast < exTimesPreFast + 8 );
			gLine.Commands.Print = TRUE;
			nextState();
			break;

		case 5:
			strcpy(txStateDesc, "Waiting the line to be printing");
			TEST_BUSY_CONDITION( gMachine.St.exec.fast < exTimesPreFast + 8 );
			TEST_BUSY_CONDITION( gLine.Status != LINE_PREPARING_PRINT );
			nextState();
			break;

		case 6:
			strcpy(txStateDesc, "Waiting the line to control stop");
			gLine.Commands.Stop = TRUE;
			TEST_BUSY_CONDITION( gLine.Status != LINE_CONTROLLED_STOP );
			nextState();
			break;

		case 7:
			strcpy(txStateDesc, "Waiting the line to be stopped");
			TEST_BUSY_CONDITION( gMachine.St.exec.fast < exTimesPreFast + 8 );
			gMachine.In.Buttons.xReset = TRUE;
			TEST_BUSY_CONDITION( gLine.Status == LINE_CONTROLLED_STOP );
			TEST_ASSERT(gLine.Status == LINE_STOPPED);

			iTestState = 0;
			TEST_DONE;

			break;

		default:
			break;
	}
}

_TEST test_ControlStopWhileStartingPrintingLine(void)
{
	if (!gMachine.Pt.xControlledByLine ){
		iTestState = 0;
		TEST_DONE;
	}
	strcpy(txTest, "test_ControlStopWhileStartingPrintingLine");
	switch (iTestState)
	{
		case 0:
			gSimMachine.Commands.xToZero = TRUE;
			nextState();
			break;

		case 1:
			strcpy(txStateDesc, "Waiting the machine to be in Zero");
			TEST_BUSY_CONDITION( gMachine.St.exec.fast < exTimesPreFast + 3 );
			TEST_BUSY_CONDITION( !gMachine.St.Mode.xZero );
			nextState();
			break;

		case 2:
			gSimMachine.Commands.xToAuto = TRUE;
			nextState();
			break;

		case 3:
			strcpy(txStateDesc, "Waiting the machine to be in Auto");
			TEST_BUSY_CONDITION( !gMachine.St.Mode.xAuto );
			gMachine.In.Buttons.xReset = TRUE;
			nextState();
			break;

		case 4:
			strcpy(txStateDesc, "Waiting the machine to be ready");
			TEST_BUSY_CONDITION( gMachine.St.exec.fast < exTimesPreFast + 8 );
			gLine.Commands.Print = TRUE;
			nextState();
			break;

		case 5:
			strcpy(txStateDesc, "Waiting the line to be printing");
			TEST_BUSY_CONDITION( gMachine.St.exec.fast < exTimesPreFast + 8 );
			TEST_BUSY_CONDITION( gLine.Status != LINE_STARTING_PRINTING );
			nextState();
			break;

		case 6:
			strcpy(txStateDesc, "Waiting the line to control stop");
			gLine.Commands.Stop = TRUE;
			TEST_BUSY_CONDITION( gLine.Status != LINE_CONTROLLED_STOP );
			TEST_ASSERT(gTransVacuum[1].Parameters.rVacPressureSetPointPerc == rPreviousVacPressureSp);
			nextState();
			break;

		case 7:
			strcpy(txStateDesc, "Waiting the line to be stopped");
			TEST_BUSY_CONDITION( gMachine.St.exec.fast < exTimesPreFast + 8 );
			gMachine.In.Buttons.xReset = TRUE;
			TEST_BUSY_CONDITION( gLine.Status == LINE_CONTROLLED_STOP );
			TEST_ASSERT(gLine.Status == LINE_STOPPED);

			iTestState = 0;
			TEST_DONE;

			break;

		default:
			break;
	}
}

_TEST test_ControlStopWhilePausingLine(void)
{
	if (!gMachine.Pt.xControlledByLine ){
		iTestState = 0;
		TEST_DONE;
	}
	strcpy(txTest, "test_ControlStopWhilePausingLine");
	switch (iTestState)
	{
		case 0:
			gSimMachine.Commands.xToZero = TRUE;
			nextState();
			break;

		case 1:
			strcpy(txStateDesc, "Waiting the machine to be in Zero");
			TEST_BUSY_CONDITION( gMachine.St.exec.fast < exTimesPreFast + 3 );
			TEST_BUSY_CONDITION( !gMachine.St.Mode.xZero );
			nextState();
			break;

		case 2:
			gSimMachine.Commands.xToAuto = TRUE;
			nextState();
			break;

		case 3:
			strcpy(txStateDesc, "Waiting the machine to be in Auto");
			TEST_BUSY_CONDITION( !gMachine.St.Mode.xAuto );
			gMachine.In.Buttons.xReset = TRUE;
			nextState();
			break;

		case 4:
			strcpy(txStateDesc, "Waiting the machine to be ready");
			TEST_BUSY_CONDITION( gMachine.St.exec.fast < exTimesPreFast + 8 );
			gLine.Commands.Print = TRUE;
			nextState();
			break;

		case 5:
			strcpy(txStateDesc, "Waiting the line to be printing");
			TEST_BUSY_CONDITION( gMachine.St.exec.fast < exTimesPreFast + 8 );
			TEST_BUSY_CONDITION( gLine.Status != LINE_PRINTING );
			nextState();
			break;

		case 6:
			strcpy(txStateDesc, "Waiting the machine to be ready");
			TEST_BUSY_CONDITION( gMachine.St.exec.fast < exTimesPreFast + 8 );
			gLine.Commands.Pause = TRUE;
			TEST_BUSY_CONDITION( gLine.Status != LINE_PAUSING );
			nextState();
			break;

		case 7:
			strcpy(txStateDesc, "Waiting the line to control stop");
			gLine.Commands.Stop = TRUE;
			TEST_BUSY_CONDITION( gLine.Status != LINE_CONTROLLED_STOP );
			nextState();
			break;

		case 8:
			strcpy(txStateDesc, "Waiting the line to be stopped");
			TEST_BUSY_CONDITION( gMachine.St.exec.fast < exTimesPreFast + 8 );
			gMachine.In.Buttons.xReset = TRUE;
			TEST_BUSY_CONDITION( gLine.Status == LINE_CONTROLLED_STOP );
			TEST_ASSERT(gLine.Status == LINE_STOPPED);

			iTestState = 0;
			TEST_DONE;

			break;

		default:
			break;
	}
}

_TEST test_CleanCommandSentWhilePausingLine(void)
{
	if (!gMachine.Pt.xControlledByLine ){
		iTestState = 0;
		TEST_DONE;
	}
	strcpy(txTest, "test_CleanCommandSentWhilePausingLine");
	switch (iTestState)
	{
		case 0:
			gSimMachine.Commands.xToZero = TRUE;
			nextState();
			break;

		case 1:
			strcpy(txStateDesc, "Waiting the machine to be in Zero");
			TEST_BUSY_CONDITION( gMachine.St.exec.fast < exTimesPreFast + 3 );
			TEST_BUSY_CONDITION( !gMachine.St.Mode.xZero );
			nextState();
			break;

		case 2:
			gSimMachine.Commands.xToAuto = TRUE;
			nextState();
			break;

		case 3:
			strcpy(txStateDesc, "Waiting the machine to be in Auto");
			TEST_BUSY_CONDITION( !gMachine.St.Mode.xAuto );
			gMachine.In.Buttons.xReset = TRUE;
			nextState();
			break;

		case 4:
			strcpy(txStateDesc, "Waiting the machine to be ready");
			TEST_BUSY_CONDITION( gMachine.St.exec.fast < exTimesPreFast + 8 );
			gLine.Commands.Print = TRUE;
			nextState();
			break;

		case 5:
			strcpy(txStateDesc, "Waiting the line to be printing");
			TEST_BUSY_CONDITION( gMachine.St.exec.fast < exTimesPreFast + 8 );
			TEST_BUSY_CONDITION( gLine.Status != LINE_PRINTING );
			nextState();
			break;

		case 6:
			strcpy(txStateDesc, "Waiting the machine to be ready");
			TEST_BUSY_CONDITION(gMachine.St.exec.fast < exTimesPreFast + 8);
			gLine.Commands.Pause = TRUE;
			TEST_BUSY_CONDITION(gLine.Status != LINE_PAUSING);
			gLine.Commands.Clean = TRUE;
			nextState();
			break;

		case 7:
			strcpy(txStateDesc, "Waiting the line to be paused");
			TEST_BUSY_CONDITION(gLine.Status != LINE_PAUSED);
			nextState();
			break;

		case 8:
			strcpy(txStateDesc, "Waiting the line to be cleaning printheads");
			TEST_BUSY_CONDITION(gLine.Status == LINE_PAUSED);
			TEST_ASSERT(gLine.StatusSummary.xCleaning);
			nextState();
			break;

		case 9:
			strcpy(txStateDesc, "Waiting the line to come back to paused");
			TEST_BUSY_CONDITION(gLine.StatusSummary.xCleaning);
			TEST_ASSERT(gLine.StatusSummary.xPausing);

			iTestState = 0;
			TEST_DONE;

			break;

		default:
			break;
	}
}

_TEST test_ControlStopWhilePausedLine(void)
{
	if (!gMachine.Pt.xControlledByLine ){
		iTestState = 0;
		TEST_DONE;
	}
	strcpy(txTest, "test_ControlStopWhilePausedLine");
	switch (iTestState)
	{
		case 0:
			gSimMachine.Commands.xToZero = TRUE;
			nextState();
			break;

		case 1:
			strcpy(txStateDesc, "Waiting the machine to be in Zero");
			TEST_BUSY_CONDITION( gMachine.St.exec.fast < exTimesPreFast + 3 );
			TEST_BUSY_CONDITION( !gMachine.St.Mode.xZero );
			nextState();
			break;

		case 2:
			gSimMachine.Commands.xToAuto = TRUE;
			nextState();
			break;

		case 3:
			strcpy(txStateDesc, "Waiting the machine to be in Auto");
			TEST_BUSY_CONDITION( !gMachine.St.Mode.xAuto );
			gMachine.In.Buttons.xReset = TRUE;
			nextState();
			break;

		case 4:
			strcpy(txStateDesc, "Waiting the machine to be ready");
			TEST_BUSY_CONDITION( gMachine.St.exec.fast < exTimesPreFast + 8 );
			gLine.Commands.Print = TRUE;
			nextState();
			break;

		case 5:
			strcpy(txStateDesc, "Waiting the line to be printing");
			TEST_BUSY_CONDITION( gMachine.St.exec.fast < exTimesPreFast + 8 );
			TEST_BUSY_CONDITION( gLine.Status != LINE_PRINTING );
			nextState();
			break;

		case 6:
			strcpy(txStateDesc, "Waiting the machine to be ready");
			TEST_BUSY_CONDITION( gMachine.St.exec.fast < exTimesPreFast + 8 );
			gLine.Commands.Pause = TRUE;
			nextState();
			break;

		case 7:
			strcpy(txStateDesc, "Waiting the machine to be ready");
			TEST_BUSY_CONDITION( gMachine.St.exec.fast < exTimesPreFast + 8 );
			TEST_BUSY_CONDITION( gLine.Status != LINE_PAUSED );
			TEST_ASSERT(gTransVacuum[1].Parameters.rVacPressureSetPointPerc < gTransVacuum[1].parSw.rVacPressureSetPointPerc);
			rPreviousVacPressureSp = gTransVacuum[1].Parameters.rVacPressureSetPointPerc;
			nextState();
			break;

		case 8:
			strcpy(txStateDesc, "Waiting the line to control stop");
			gLine.Commands.Stop = TRUE;
			TEST_BUSY_CONDITION( gLine.Status != LINE_CONTROLLED_STOP );
			nextState();
			break;

		case 9:
			strcpy(txStateDesc, "Waiting the line to be stopped");
			TEST_BUSY_CONDITION( gMachine.St.exec.fast < exTimesPreFast + 8 );
			gMachine.In.Buttons.xReset = TRUE;
			TEST_BUSY_CONDITION( gLine.Status == LINE_CONTROLLED_STOP );
			TEST_ASSERT(gLine.Status == LINE_STOPPED);

			iTestState = 0;
			TEST_DONE;

			break;

		default:
			break;
	}
}

_TEST test_ControlStopWhileBeltEmptyingLine(void)
{
	if (!gMachine.Pt.xControlledByLine ){
		iTestState = 0;
		TEST_DONE;
	}
	strcpy(txTest, "test_ControlStopWhileBeltEmptyingLine");
	switch (iTestState)
	{
		case 0:
			gSimMachine.Commands.xToZero = TRUE;
			gMachine.parSw.rBeltSpeedSetPoint = gMachine.Pt.rBeltSpeedWhileEmptyBelt + 20.0;
			nextState();
			break;

		case 1:
			strcpy(txStateDesc, "Waiting the machine to be in Zero");
			TEST_BUSY_CONDITION( gMachine.St.exec.fast < exTimesPreFast + 3 );
			TEST_BUSY_CONDITION( !gMachine.St.Mode.xZero );
			nextState();
			break;

		case 2:
			gSimMachine.Commands.xToAuto = TRUE;
			nextState();
			break;

		case 3:
			strcpy(txStateDesc, "Waiting the machine to be in Auto");
			TEST_BUSY_CONDITION( !gMachine.St.Mode.xAuto );
			gMachine.In.Buttons.xReset = TRUE;
			nextState();
			break;

		case 4:
			strcpy(txStateDesc, "Waiting the machine to be ready");
			TEST_BUSY_CONDITION( gMachine.St.exec.fast < exTimesPreFast + 8 );
			gLine.Commands.Print = TRUE;
			nextState();
			break;

		case 5:
			strcpy(txStateDesc, "Waiting the line to be printing");
			TEST_BUSY_CONDITION( gMachine.St.exec.fast < exTimesPreFast + 8 );
			TEST_BUSY_CONDITION( gLine.Status != LINE_PRINTING );
			if (gCuringLed[iIndexColorCuringLedBar].Status.xInstalled){
				TEST_BUSY_CONDITION( !gCuringLed[iIndexColorCuringLedBar].Status.xEmitting );
			}
			nextState();
			break;

		case 6:
			gSimMachine.Commands.xToZero = TRUE;
			TEST_BUSY_CONDITION( !gMachine.St.Mode.xZero );
			nextState();
			break;

		case 7:
			gSimMachine.Commands.xToAuto = TRUE;
			nextState();
			break;

		case 8:
			strcpy(txStateDesc, "Waiting the machine to be in Auto");
			TEST_BUSY_CONDITION( !gMachine.St.Mode.xAuto );
			gMachine.In.Buttons.xReset = TRUE;
			nextState();
			break;

		case 9:
			strcpy(txStateDesc, "Waiting the machine to be ready");
			TEST_BUSY_CONDITION( gMachine.St.exec.fast < exTimesPreFast + 8 );
			gLine.Commands.EmptyBelt = TRUE;
			nextState();
			break;

		case 10:
			strcpy(txStateDesc, "Waiting the line to be emptying belts");
			TEST_BUSY_CONDITION( gMachine.St.exec.fast < exTimesPreFast + 8 );
			TEST_BUSY_CONDITION( gLine.Status != LINE_BELT_EMPTYING );
			TEST_ASSERT(gBelt.parameters.rSetPointSpeed == gMachine.Pt.rBeltSpeedWhileEmptyBelt);
			TEST_ASSERT(gBelt.parameters.rSetPointSpeed != gMachine.parSw.rBeltSpeedSetPoint);
			TEST_ASSERT(gTransVacuum[1].Parameters.rVacPressureSetPointPerc > gTransVacuum[1].parSw.rVacPressureSetPointPerc);
			rPreviousVacPressureSp = gTransVacuum[1].Parameters.rVacPressureSetPointPerc;
			nextState();
			break;

		case 11:
			strcpy(txStateDesc, "Waiting the line to control stop");
			gLine.Commands.Stop = TRUE;
			TEST_BUSY_CONDITION( gLine.Status != LINE_CONTROLLED_STOP );
			TEST_ASSERT(gTransVacuum[1].Parameters.rVacPressureSetPointPerc == rPreviousVacPressureSp);
			nextState();
			break;

		case 12:
			strcpy(txStateDesc, "Waiting the line to be stopped");
			TEST_BUSY_CONDITION( gMachine.St.exec.fast < exTimesPreFast + 8 );
			gMachine.In.Buttons.xReset = TRUE;
			TEST_BUSY_CONDITION( gLine.Status == LINE_CONTROLLED_STOP );
			TEST_ASSERT(gLine.Status == LINE_STOPPED);
			nextState();
			break;

		case 13:
			strcpy(txStateDesc, "Waiting the line to be idle");
			TEST_BUSY_CONDITION( gLine.Status != LINE_IDLE );
			nextState();
			break;

		case 14:
			strcpy(txStateDesc, "Waiting the Clean order signal");

			iTestState = 0;
			TEST_DONE;

			break;

		default:
			break;
	}
}

_TEST test_ControlStopWhilePrepareToEmptyBeltLine(void)
{
	if (!gMachine.Pt.xControlledByLine ){
		iTestState = 0;
		TEST_DONE;
	}
	strcpy(txTest, "test_ControlStopWhilePrepareToEmptyBeltLine");
	switch (iTestState)
	{
		case 0:
			gSimMachine.Commands.xToZero = TRUE;
			nextState();
			break;

		case 1:
			strcpy(txStateDesc, "Waiting the machine to be in Zero");
			TEST_BUSY_CONDITION( gMachine.St.exec.fast < exTimesPreFast + 3 );
			TEST_BUSY_CONDITION( !gMachine.St.Mode.xZero );
			nextState();
			break;

		case 2:
			gSimMachine.Commands.xToAuto = TRUE;
			nextState();
			break;

		case 3:
			strcpy(txStateDesc, "Waiting the machine to be in Auto");
			TEST_BUSY_CONDITION( !gMachine.St.Mode.xAuto );
			gMachine.In.Buttons.xReset = TRUE;
			nextState();
			break;

		case 4:
			strcpy(txStateDesc, "Waiting the machine to be ready");
			TEST_BUSY_CONDITION( gMachine.St.exec.fast < exTimesPreFast + 8 );
			gLine.Commands.EmptyBelt = TRUE;
			TEST_BUSY_CONDITION( gLine.Status != LINE_PREPARING_EMPTYBELT );
			nextState();
			break;

		case 5:
			strcpy(txStateDesc, "Waiting the line to control stop");
			gLine.Commands.Stop = TRUE;
			TEST_BUSY_CONDITION( gLine.Status != LINE_CONTROLLED_STOP );
			nextState();
			break;

		case 6:
			strcpy(txStateDesc, "Waiting the line to be stopped");
			TEST_BUSY_CONDITION( gMachine.St.exec.fast < exTimesPreFast + 8 );
			gMachine.In.Buttons.xReset = TRUE;
			TEST_BUSY_CONDITION( gLine.Status == LINE_CONTROLLED_STOP );
			TEST_ASSERT(gLine.Status == LINE_STOPPED);

			iTestState = 0;
			TEST_DONE;

			break;

		default:
			break;
	}
}

_TEST test_ControlStopWhileStartingEmptyBeltLine(void)
{
	if (!gMachine.Pt.xControlledByLine ){
		iTestState = 0;
		TEST_DONE;
	}
	strcpy(txTest, "test_ControlStopWhileStartingEmptyBeltLine");
	switch (iTestState)
	{
		case 0:
			gFeeder.ParSw.xEnabled=FALSE; //Disabling feeder to not active virtual media in SimMachine
			gSimMachine.Commands.xToZero = TRUE;
			nextState();
			break;

		case 1:
			strcpy(txStateDesc, "Waiting the machine to be in Zero");
			TEST_BUSY_CONDITION( gMachine.St.exec.fast < exTimesPreFast + 3 );
			TEST_BUSY_CONDITION( !gMachine.St.Mode.xZero );
			nextState();
			break;

		case 2:
			gSimMachine.Commands.xToAuto = TRUE;
			nextState();
			break;

		case 3:
			strcpy(txStateDesc, "Waiting the machine to be in Auto");
			TEST_BUSY_CONDITION( !gMachine.St.Mode.xAuto );
			gMachine.In.Buttons.xReset = TRUE;
			nextState();
			break;

		case 4:
			strcpy(txStateDesc, "Waiting the machine to be ready");
			TEST_BUSY_CONDITION( gMachine.St.exec.fast < exTimesPreFast + 8 );
			gLine.Commands.EmptyBelt = TRUE;
			nextState();
			break;

		case 5:
			strcpy(txStateDesc, "Waiting the line to start empty belt");
			TEST_BUSY_CONDITION( gLine.Status != LINE_STARTING_EMPTYBELT );
			nextState();
			break;

		case 6:
			strcpy(txStateDesc, "Waiting the line to control stop");
			TEST_BUSY_CONDITION( gLine.Status != LINE_CONTROLLED_STOP );
			nextState();
			break;

		case 7:
			strcpy(txStateDesc, "Waiting the line to be stopped");
			TEST_BUSY_CONDITION( gMachine.St.exec.fast < exTimesPreFast + 8 );
			gMachine.In.Buttons.xReset = TRUE;
			TEST_BUSY_CONDITION( gLine.Status == LINE_CONTROLLED_STOP );
			TEST_ASSERT(gLine.Status == LINE_STOPPED);
			gFeeder.ParSw.xEnabled=TRUE; //Enabling feeder again to use it in next tests
			iTestState = 0;
			TEST_DONE;

			break;

		default:
			break;
	}
}

_TEST test_ControlStopWhileCleaningLine(void)
{
	if (!gMachine.Pt.xControlledByLine ){
		iTestState = 0;
		TEST_DONE;
	}
	strcpy(txTest, "test_ControlStopWhileCleaningLine");
	switch (iTestState)
	{
		case 0:
			gSimMachine.Commands.xToZero = TRUE;
			nextState();
			break;

		case 1:
			strcpy(txStateDesc, "Waiting the machine to be in Zero");
			TEST_BUSY_CONDITION( gMachine.St.exec.fast < exTimesPreFast + 3 );
			TEST_BUSY_CONDITION( !gMachine.St.Mode.xZero );
			nextState();
			break;

		case 2:
			gSimMachine.Commands.xToAuto = TRUE;
			nextState();
			break;

		case 3:
			strcpy(txStateDesc, "Waiting the machine to be in Auto");
			TEST_BUSY_CONDITION( !gMachine.St.Mode.xAuto );
			gMachine.In.Buttons.xReset = TRUE;
			nextState();
			break;

		case 4:
			strcpy(txStateDesc, "Waiting the machine to be ready");
			TEST_BUSY_CONDITION( gMachine.St.exec.fast < exTimesPreFast + 8 );
			gLine.Commands.Print = TRUE;
			nextState();
			break;

		case 5:
			strcpy(txStateDesc, "Waiting the line to be printing");
			TEST_BUSY_CONDITION( gMachine.St.exec.fast < exTimesPreFast + 8 );
			TEST_BUSY_CONDITION( gLine.Status != LINE_PRINTING );
			nextState();
			break;

		case 6:
			strcpy(txStateDesc, "Waiting the machine to be ready");
			TEST_BUSY_CONDITION( gMachine.St.exec.fast < exTimesPreFast + 8 );
			gLine.Commands.Clean = TRUE;
			nextState();
			break;

		case 7:
			strcpy(txStateDesc, "Waiting the line to be emptying belts");
			TEST_BUSY_CONDITION( gMachine.St.exec.fast < exTimesPreFast + 8 );
			TEST_BUSY_CONDITION( gLine.Status != LINE_CLEANINGPH );
			nextState();
			break;

		case 8:
			strcpy(txStateDesc, "Waiting the line to control stop");
			gLine.Commands.Stop = TRUE;
			TEST_BUSY_CONDITION( gLine.Status != LINE_CONTROLLED_STOP );
			nextState();
			break;

		case 9:
			strcpy(txStateDesc, "Waiting the line to be stopped");
			TEST_BUSY_CONDITION( gMachine.St.exec.fast < exTimesPreFast + 8 );
			gMachine.In.Buttons.xReset = TRUE;
			TEST_BUSY_CONDITION( gLine.Status == LINE_CONTROLLED_STOP );
			TEST_ASSERT(gLine.Status == LINE_STOPPED);

			iTestState = 0;
			TEST_DONE;

			break;

		default:
			break;
	}
}

_TEST test_ControlStopWhilePrepareToCleanLine(void)
{
	if (!gMachine.Pt.xControlledByLine ){
		iTestState = 0;
		TEST_DONE;
	}
	strcpy(txTest, "test_ControlStopWhilePrepareToCleanLine");
	switch (iTestState)
	{
		case 0:
			gSimMachine.Commands.xToZero = TRUE;
			nextState();
			break;

		case 1:
			strcpy(txStateDesc, "Waiting the machine to be in Zero");
			TEST_BUSY_CONDITION( gMachine.St.exec.fast < exTimesPreFast + 3 );
			TEST_BUSY_CONDITION( !gMachine.St.Mode.xZero );
			nextState();
			break;

		case 2:
			gSimMachine.Commands.xToAuto = TRUE;
			nextState();
			break;

		case 3:
			strcpy(txStateDesc, "Waiting the machine to be in Auto");
			TEST_BUSY_CONDITION( !gMachine.St.Mode.xAuto );
			gMachine.In.Buttons.xReset = TRUE;
			nextState();
			break;

		case 4:
			strcpy(txStateDesc, "Waiting the machine to be ready");
			TEST_BUSY_CONDITION( gMachine.St.exec.fast < exTimesPreFast + 8 );
			gLine.Commands.Print = TRUE;
			nextState();
			break;

		case 5:
			strcpy(txStateDesc, "Waiting the line to be printing");
			TEST_BUSY_CONDITION( gMachine.St.exec.fast < exTimesPreFast + 8 );
			TEST_BUSY_CONDITION( gLine.Status != LINE_PRINTING );
			nextState();
			break;

		case 6:
			strcpy(txStateDesc, "Waiting the machine to be ready");
			TEST_BUSY_CONDITION( gMachine.St.exec.fast < exTimesPreFast + 8 );
			gLine.Commands.Clean = TRUE;
			nextState();
			break;

		case 7:
			strcpy(txStateDesc, "Waiting the line to prepare to clean");
			TEST_BUSY_CONDITION( gLine.Status != LINE_PREPARING_CLEANPH );
			gLine.Commands.Stop = TRUE;
			nextState();
			break;

		case 8:
			strcpy(txStateDesc, "Waiting the line to control stop");
			TEST_BUSY_CONDITION( gLine.Status != LINE_CONTROLLED_STOP );
			nextState();
			break;

		case 9:
			strcpy(txStateDesc, "Waiting the line to be stopped");
			TEST_BUSY_CONDITION( gMachine.St.exec.fast < exTimesPreFast + 8 );
			gMachine.In.Buttons.xReset = TRUE;
			TEST_BUSY_CONDITION( gLine.Status == LINE_CONTROLLED_STOP );
			TEST_ASSERT(gLine.Status == LINE_STOPPED);
			nextState();
			break;

		case 10:
			strcpy(txStateDesc, "Waiting the machine to be start cleaning");
			gSimMachine.Commands.xToAuto = TRUE;
			gMachine.In.Buttons.xReset = TRUE;
			TEST_BUSY_CONDITION( !gMachine.St.Mode.xAuto );
			TEST_BUSY_CONDITION( gLine.Status != LINE_STARTING_CLEANINGPH );
			iTestState = 0;
			TEST_DONE;

		default:
			break;
	}
}

_TEST test_ControlStopWhileStartingCleaningLine(void)
{
	if (!gMachine.Pt.xControlledByLine){
		iTestState = 0;
		TEST_DONE;
	}
	strcpy(txTest, "test_ControlStopWhileStartingCleaningLine");
	switch (iTestState)
	{
		case 0:
			gSimMachine.Commands.xToZero = TRUE;
			nextState();
			break;

		case 1:
			strcpy(txStateDesc, "Waiting the machine to be in Zero");
			TEST_BUSY_CONDITION( gMachine.St.exec.fast < exTimesPreFast + 3 );
			TEST_BUSY_CONDITION( !gMachine.St.Mode.xZero );
			nextState();
			break;

		case 2:
			gSimMachine.Commands.xToAuto = TRUE;
			nextState();
			break;

		case 3:
			strcpy(txStateDesc, "Waiting the machine to be in Auto");
			TEST_BUSY_CONDITION( !gMachine.St.Mode.xAuto );
			gMachine.In.Buttons.xReset = TRUE;
			nextState();
			break;

		case 4:
			strcpy(txStateDesc, "Waiting the machine to be ready");
			TEST_BUSY_CONDITION( gMachine.St.exec.fast < exTimesPreFast + 8 );
			TEST_BUSY_CONDITION( gLine.Status != LINE_IDLE );
			gLine.Commands.Print = TRUE;
			nextState();
			break;

		case 5:
			strcpy(txStateDesc, "Waiting the line to be printing");
			TEST_BUSY_CONDITION( gMachine.St.exec.fast < exTimesPreFast + 8 );
			TEST_BUSY_CONDITION( gLine.Status != LINE_PRINTING );
			nextState();
			break;

		case 6:
			strcpy(txStateDesc, "Waiting the machine to be ready");
			TEST_BUSY_CONDITION( gMachine.St.exec.fast < exTimesPreFast + 8 );
			gLine.Commands.Clean = TRUE;
			nextState();
			break;

		case 7:
			strcpy(txStateDesc, "Waiting the line to start empty belt");
			TEST_BUSY_CONDITION( gMachine.St.exec.fast < exTimesPreFast + 8 );
			TEST_BUSY_CONDITION( gLine.Status != LINE_STARTING_CLEANINGPH );
			nextState();
			break;

		case 8:
			strcpy(txStateDesc, "Waiting the line to control stop");
			gLine.Commands.Stop = TRUE;
			TEST_BUSY_CONDITION( gLine.Status != LINE_CONTROLLED_STOP );
			nextState();
			break;

		case 9:
			strcpy(txStateDesc, "Waiting the line to be stopped");
			TEST_BUSY_CONDITION( gMachine.St.exec.fast < exTimesPreFast + 8 );
			gMachine.In.Buttons.xReset = TRUE;
			TEST_BUSY_CONDITION( gLine.Status == LINE_CONTROLLED_STOP );
			TEST_ASSERT(gLine.Status == LINE_STOPPED);

			iTestState = 0;
			TEST_DONE;

			break;

		default:
			break;
	}
}

_TEST test_CriticalAlarmWhilePrintingLine(void)
{
	if (!gMachine.Pt.xControlledByLine){
		iTestState = 0;
		TEST_DONE;
	}
	strcpy(txTest, "test_CriticalAlarmWhilePrintingLine");
	switch (iTestState)
	{
		case 0:
			gSimMachine.Commands.xToZero = TRUE;
			nextState();
			break;

		case 1:
			strcpy(txStateDesc, "Waiting the machine to be in Zero");
			TEST_BUSY_CONDITION( gMachine.St.exec.fast < exTimesPreFast + 3 );
			TEST_BUSY_CONDITION( !gMachine.St.Mode.xZero );
			nextState();
			break;

		case 2:
			gSimMachine.Commands.xToAuto = TRUE;
			nextState();
			break;

		case 3:
			strcpy(txStateDesc, "Waiting the machine to be in Auto");
			TEST_BUSY_CONDITION( gLine.Status !=  LINE_IDLE );
			nextState();
			break;

		case 4:
			strcpy(txStateDesc, "Waiting the machine to be ready");
			TEST_BUSY_CONDITION( gMachine.St.exec.fast < exTimesPreFast + 8 );
			gLine.Commands.Print = TRUE;
			nextState();
			break;

		case 5:
			strcpy(txStateDesc, "Waiting the line to start printing");
			TEST_BUSY_CONDITION( gMachine.St.exec.fast < exTimesPreFast + 8 );
			TEST_BUSY_CONDITION( gLine.Status != LINE_PRINTING );
			nextState();
			break;

		case 6:
			strcpy(txStateDesc, "Waiting the line to stop");
			gMachine.In.xPowerSwitch=FALSE;
			TEST_BUSY_CONDITION( gLine.Status != LINE_ERROR);
			TEST_ASSERT(gMachine.Al.Alarm.xNoPowered);
			TEST_ASSERT(gMachine.AlSummary.xAlarmCritical);
			gMachine.In.xPowerSwitch=TRUE;
			nextState();
			break;

		case 7:
			strcpy(txStateDesc, "Waiting the line to control stop");
			TEST_BUSY_CONDITION( gMachine.St.exec.fast < exTimesPreFast + 8 );
			gMachine.In.Buttons.xReset = TRUE;
			gSimMachine.Commands.xToZero = TRUE;
			TEST_BUSY_CONDITION( !gMachine.St.Mode.xZero );
			gSimMachine.Commands.xToAuto = TRUE;
			gMachine.In.Buttons.xReset = TRUE;
			nextState();
			break;

		case 8:
			strcpy(txStateDesc, "Waiting the line to be stopped");
			TEST_BUSY_CONDITION( gMachine.St.exec.fast < exTimesPreFast + 8 );
			TEST_BUSY_CONDITION( gLine.Status != LINE_IDLE );
			TEST_ASSERT(gLine.Status == LINE_IDLE);

			iTestState = 0;
			TEST_DONE;

			break;

		default:
			break;
	}
}

_TEST test_CriticalAlarmDueToEhdJamAlarm(void)
{
	if (!gEdgeHoldDown.parameters.xInstalled || TRUE){
		TEST_DONE;
	}

	if (!gMachine.Pt.xControlledByLine ){
		iTestState = 0;
		TEST_DONE;
	}
	strcpy(txTest, "test_CriticalAlarmDueToEhdJamAlarm");
	switch (iTestState)
	{
		case 0:
			gSimMachine.Commands.xToZero = TRUE;
			nextState();
			break;

		case 1:
			strcpy(txStateDesc, "Waiting the machine to be in Zero");
			TEST_BUSY_CONDITION( gMachine.St.exec.fast < exTimesPreFast + 3 );
			TEST_BUSY_CONDITION( !gMachine.St.Mode.xZero );
			nextState();
			break;

		case 2:
			gSimMachine.Commands.xToAuto = TRUE;
			nextState();
			break;

		case 3:
			strcpy(txStateDesc, "Waiting the machine to be in Auto");
			TEST_BUSY_CONDITION( gLine.Status !=  LINE_IDLE );
			nextState();
			break;

		case 4:
			strcpy(txStateDesc, "Waiting the machine to be ready");
			TEST_BUSY_CONDITION( gMachine.St.exec.fast < exTimesPreFast + 8 );
			gLine.Commands.Print = TRUE;
			nextState();
			break;

		case 5:
			strcpy(txStateDesc, "Waiting the line to start printing");
			TEST_BUSY_CONDITION( gMachine.St.exec.fast < exTimesPreFast + 8 );
			TEST_BUSY_CONDITION( gLine.Status != LINE_PRINTING );
			nextState();
			break;

		case 6:
			strcpy(txStateDesc, "Waiting the line to stop");
			gEdgeHoldDown.Alarms.xJam = TRUE;
			TEST_BUSY_CONDITION( gLine.Status != LINE_ERROR);
			nextState();
			break;

		case 7:
			strcpy(txStateDesc, "Waiting the line to control stop");
			gMachine.In.Buttons.xReset = TRUE;
			TEST_BUSY_CONDITION( gMachine.St.exec.fast < exTimesPreFast + 8 );
			gSimMachine.Commands.xToZero = TRUE;
			TEST_BUSY_CONDITION( !gMachine.St.Mode.xZero );
			gSimMachine.Commands.xToAuto = TRUE;
			gMachine.In.Buttons.xReset = TRUE;
			nextState();
			break;

		case 8:
			strcpy(txStateDesc, "Waiting the line to be stopped");
			TEST_BUSY_CONDITION( gMachine.St.exec.fast < exTimesPreFast + 8 );
			TEST_BUSY_CONDITION( gLine.Status != LINE_IDLE );
			TEST_ASSERT(gLine.Status == LINE_IDLE);

			iTestState = 0;
			TEST_DONE;

			break;

		default:
			break;
	}
}

_TEST test_EhdGoesToResetPositionWhenDisabled(void)
{
	if (!gEdgeHoldDown.parameters.xInstalled || TRUE){
		TEST_DONE;
	}

	if (!gMachine.Pt.xControlledByLine ){
		iTestState = 0;
		TEST_DONE;
	}
	strcpy(txTest, "test_EhdGoesToResetPositionWhenDisabled");
	switch (iTestState)
	{
		case 0:
			gSimMachine.Commands.xToZero = TRUE;
			nextState();
			break;

		case 1:
			strcpy(txStateDesc, "Waiting the machine to be in Zero");
			TEST_BUSY_CONDITION( gMachine.St.exec.fast < exTimesPreFast + 3 );
			TEST_BUSY_CONDITION( !gMachine.St.Mode.xZero );
			nextState();
			break;

		case 2:
			gSimMachine.Commands.xToAuto = TRUE;
			nextState();
			break;

		case 3:
			strcpy(txStateDesc, "Waiting the machine to be in Auto");
			TEST_BUSY_CONDITION( gLine.Status !=  LINE_IDLE );
			nextState();
			break;

		case 4:
			strcpy(txStateDesc, "Waiting the machine to be ready");
			TEST_BUSY_CONDITION( gMachine.St.exec.fast < exTimesPreFast + 8 );
			gLine.Commands.Print = TRUE;
			nextState();
			break;

		case 5:
			strcpy(txStateDesc, "Waiting the line to start printing");
			TEST_BUSY_CONDITION( gMachine.St.exec.fast < exTimesPreFast + 8 );
			TEST_BUSY_CONDITION( gLine.Status != LINE_PRINTING );
			nextState();
			break;

		case 6:
			strcpy(txStateDesc, "Going to zero state");
			gSimMachine.Commands.xToZero = TRUE;
			TEST_BUSY_CONDITION( !gMachine.St.Mode.xZero );
			nextState();
			break;

		case 7:
			strcpy(txStateDesc, "Entering auto again");
			//gEdgeHoldDown.parSw.xEnable = FALSE;
			gSimMachine.Commands.xToAuto = TRUE;
			gMachine.In.Buttons.xReset = TRUE;
			TEST_BUSY_CONDITION( !gMachine.St.Mode.xAuto );
			TEST_ASSERT(gEdgeHoldDown.status.xEnabled);
			if(gCuringLed[iIndexColorCuringLedBar].Status.xInstalled){
				TEST_ASSERT(gCuringLed[iIndexColorCuringLedBar].Parameters.xCureByStretch);
				TEST_ASSERT(gCuringLed[iIndexColorCuringLedBar].Parameters.xOptimizeCuring);
			}
			nextState();
			break;

		case 8:
			strcpy(txStateDesc, "Waiting the ehd to go to reset position");
			TEST_BUSY_CONDITION( gMachine.St.exec.fast < exTimesPreFast + 8 );
			TEST_BUSY_CONDITION( gLine.Status != LINE_IDLE );
			TEST_BUSY_CONDITION( !gEdgeHoldDown.status.xInRestingPosition );
			nextState();
			break;

		case 9:
			strcpy(txStateDesc, "Waiting the line to be stopped");
			TEST_BUSY_CONDITION( gEdgeHoldDown.status.iSystemState!=EHD_STOPPED );
			TEST_ASSERT(!gEdgeHoldDown.status.xEnabled);
			TEST_BUSY_CONDITION( gCuringLed[iIndexColorCuringLedBar].Parameters.xCureByStretch );
			if(gCuringLed[iIndexColorCuringLedBar].Status.xInstalled && !gMachine.parSw.Curing.xCureByStretch){
				TEST_ASSERT(!gCuringLed[iIndexColorCuringLedBar].Parameters.xCureByStretch);
			}
			//gEdgeHoldDown.parSw.xEnable = TRUE;

			iTestState = 0;
			TEST_DONE;

			break;

		default:
			break;
	}
}

_TEST test_JobNotLoadedWhilePrintingLine(void)
{
	if (!gMachine.Pt.xControlledByLine ){
		iTestState = 0;
		TEST_DONE;
	}
	strcpy(txTest, "test_JobNotLoadedWhilePrintingLine");
	switch (iTestState)
	{
		case 0:
			gSimMachine.Commands.xToZero = TRUE;
			nextState();
			break;

		case 1:
			strcpy(txStateDesc, "Waiting the machine to be in Zero");
			TEST_BUSY_CONDITION( gMachine.St.exec.fast < exTimesPreFast + 3 );
			gSimThickCtrl.Commands.xEmptyMediaTracking = TRUE;
			TEST_BUSY_CONDITION( !gMachine.St.Mode.xZero );
			nextState();
			break;

		case 2:
			gSimMachine.Commands.xToAuto = TRUE;
			nextState();
			break;

		case 3:
			strcpy(txStateDesc, "Waiting the machine to be in Auto");
			TEST_BUSY_CONDITION( gLine.Status !=  LINE_IDLE );
			nextState();
			break;

		case 4:
			strcpy(txStateDesc, "Waiting the machine to be ready");
			TEST_BUSY_CONDITION( gMachine.St.exec.fast < exTimesPreFast + 8 );
			gLine.Commands.Print = TRUE;
			nextState();
			break;

		case 5:
			strcpy(txStateDesc, "Waiting the line to start printing");
			TEST_BUSY_CONDITION( gMachine.St.exec.fast < exTimesPreFast + 8 );
			TEST_BUSY_CONDITION( gLine.Status != LINE_PRINTING );
			gSimMachine.Commands.Media.xContinuousMediaPresent = TRUE;
			nextState();
			break;

		case 6:
			strcpy(txStateDesc, "Waiting the line to stop");
			gMachine.parSw.Electronics.xRobotReadyL1 =FALSE;
			TEST_BUSY_CONDITION(gLine.Status != LINE_ERROR && gLine.Status != LINE_STOPPED);
			TEST_ASSERT(gMachine.Al.Alarm.xNotLoadedImage);
			gSimMachine.Commands.Media.xContinuousMediaPresent = FALSE;
			gMachine.parSw.Electronics.xRobotReadyL1 =TRUE;
			nextState();
			break;

		case 7:
			strcpy(txStateDesc, "Waiting the line to control stop");
			TEST_BUSY_CONDITION( gMachine.St.exec.fast < exTimesPreFast + 8 );
			gMachine.In.Buttons.xReset = TRUE;
			gSimMachine.Commands.xToZero = TRUE;
			TEST_BUSY_CONDITION(!gMachine.St.Mode.xZero);
			gSimMachine.Commands.xToAuto = TRUE;
			gMachine.In.Buttons.xReset = TRUE;
			nextState();
			break;

		case 8:
			strcpy(txStateDesc, "Waiting the line to be stopped");
			TEST_BUSY_CONDITION( gMachine.St.exec.fast < exTimesPreFast + 8 );
			TEST_BUSY_CONDITION( gLine.Status != LINE_IDLE );
			TEST_ASSERT(gLine.Status == LINE_IDLE);

			iTestState = 0;
			TEST_DONE;

			break;

		default:
			break;
	}
}

_TEST test_JobNotLoadedWhilePrintingAndLineIsEmpty(void)
{

	if (!gMachine.Pt.xControlledByLine ){
		iTestState = 0;
		TEST_DONE;
	}
	strcpy(txTest, "test_JobNotLoadedWhilePrintingAndLineIsEmpty");
	switch (iTestState)
	{
		case 0:
			gSimMachine.Commands.xToZero = TRUE;
			gSimMachine.Commands.Media.xMediaIfFeederFeeding = FALSE;
			nextState();
			break;

		case 1:
			strcpy(txStateDesc, "Waiting the machine to be in Zero");
			TEST_BUSY_CONDITION( gMachine.St.exec.fast < exTimesPreFast + 3 );
			gSimThickCtrl.Commands.xEmptyMediaTracking = TRUE;
			TEST_BUSY_CONDITION( !gMachine.St.Mode.xZero );
			nextState();
			break;

		case 2:
			gSimMachine.Commands.xToAuto = TRUE;
			nextState();
			break;

		case 3:
			strcpy(txStateDesc, "Waiting the machine to be in Auto");
			TEST_BUSY_CONDITION( gLine.Status !=  LINE_IDLE );
			nextState();
			break;

		case 4:
			strcpy(txStateDesc, "Waiting the machine to be ready");
			TEST_BUSY_CONDITION( gMachine.St.exec.fast < exTimesPreFast + 8 );
			gLine.Commands.Print = TRUE;
			nextState();
			break;

		case 5:
			strcpy(txStateDesc, "Waiting the line to start printing");
			TEST_BUSY_CONDITION( gMachine.St.exec.fast < exTimesPreFast + 8 );
			TEST_BUSY_CONDITION( gLine.Status != LINE_PRINTING );
			nextState();
			break;

		case 6:
			strcpy(txStateDesc, "Waiting the line to stop");
			TEST_BUSY_CONDITION( !gThicknessCtrl.status.Belt.xBeltEmpty );
			gMachine.parSw.Electronics.xRobotReadyL1=FALSE;
			TEST_BUSY_CONDITION( gLine.Status != LINE_PAUSED);
			TEST_ASSERT(gLine.Status == LINE_PAUSED);
			if (gEdgeHoldDown.parSw.xEnable ){
				TEST_BUSY_CONDITION(!gEdgeHoldDown.parameters.xEnableMovements);
				TEST_ASSERT(gEdgeHoldDown.parameters.xEnableMovements);
				TEST_ASSERT(gBlock[1].commands.xForcePreprintingPos);
			}
			gMachine.parSw.Electronics.xRobotReadyL1 =TRUE;
			nextState();
			break;

		case 7:
			strcpy(txStateDesc, "Waiting the line to control stop");
			TEST_BUSY_CONDITION( gMachine.St.exec.fast < exTimesPreFast + 8 );
			gMachine.In.Buttons.xReset = TRUE;
			gSimMachine.Commands.xToZero = TRUE;
			TEST_BUSY_CONDITION( !gMachine.St.Mode.xZero );
			gSimMachine.Commands.xToAuto = TRUE;
			gMachine.In.Buttons.xReset = TRUE;
			nextState();
			break;

		case 8:
			strcpy(txStateDesc, "Waiting the line to be stopped");
			TEST_BUSY_CONDITION( gMachine.St.exec.fast < exTimesPreFast + 8 );
			TEST_BUSY_CONDITION( gLine.Status != LINE_IDLE );
			TEST_ASSERT(gLine.Status == LINE_IDLE);
			if (gEdgeHoldDown.parSw.xEnable ){
				TEST_ASSERT(gEdgeHoldDown.status.iSystemState==EHD_IDLE);
			}

			iTestState = 0;
			TEST_DONE;

			break;

		default:
			break;
	}
}

_TEST test_CriticalAlarmDueToDryerNotInRemoteWhilePrintingLine(void)
{
	if (!gMachine.Pt.xControlledByLine || !gDryerAnc.Parameters.xInstalled ){
		iTestState = 0;
		TEST_DONE;
	}
	strcpy(txTest, "test_CriticalAlarmDueToDryerNotInRemoteWhilePrintingLine");
	switch (iTestState)
	{
		case 0:
			gSimMachine.Commands.xToZero = TRUE;
			nextState();
			break;

		case 1:
			strcpy(txStateDesc, "Waiting the machine to be in Zero");
			TEST_BUSY_CONDITION( gMachine.St.exec.fast < exTimesPreFast + 3 );
			TEST_BUSY_CONDITION( !gMachine.St.Mode.xZero );
			nextState();
			break;

		case 2:
			gSimMachine.Commands.xToAuto = TRUE;
			nextState();
			break;

		case 3:
			strcpy(txStateDesc, "Waiting the machine to be in Auto");
			TEST_BUSY_CONDITION( gLine.Status !=  LINE_IDLE );
			nextState();
			break;

		case 4:
			strcpy(txStateDesc, "Waiting the machine to be ready");
			TEST_BUSY_CONDITION( gMachine.St.exec.fast < exTimesPreFast + 8 );
			gLine.Commands.Print = TRUE;
			nextState();
			break;

		case 5:
			strcpy(txStateDesc, "Waiting the line to start printing");
			TEST_BUSY_CONDITION( gMachine.St.exec.fast < exTimesPreFast + 8 );
			TEST_BUSY_CONDITION( gLine.Status != LINE_PRINTING );
			nextState();
			break;

		case 6:
			strcpy(txStateDesc, "Waiting the line to stop");
			gDryerAnc.Inputs.xInRemote=FALSE;
			TEST_BUSY_CONDITION( gLine.Status != LINE_ERROR );
			gDryerAnc.Inputs.xInRemote=TRUE;
			nextState();
			break;

		case 7:
			strcpy(txStateDesc, "Waiting the line to control stop");
			gMachine.In.Buttons.xReset = TRUE;
			TEST_BUSY_CONDITION( gMachine.St.exec.fast < exTimesPreFast + 8 );
			gSimMachine.Commands.xToZero = TRUE;
			TEST_BUSY_CONDITION( !gMachine.St.Mode.xZero );
			gSimMachine.Commands.xToAuto = TRUE;
			gMachine.In.Buttons.xReset = TRUE;
			nextState();
			break;

		case 8:
			strcpy(txStateDesc, "Waiting the line to be stopped");
			TEST_BUSY_CONDITION( gMachine.St.exec.fast < exTimesPreFast + 8 );
			TEST_BUSY_CONDITION( gLine.Status != LINE_IDLE );
			TEST_ASSERT(gLine.Status == LINE_IDLE);

			iTestState = 0;
			TEST_DONE;

			break;

		default:
			break;
	}
}

_TEST test_CriticalAlarmDueDryerStopButtonPressed(void)
{
	if (!gMachine.Pt.xControlledByLine || !gDryerAnc.Parameters.xInstalled ){
		iTestState = 0;
		TEST_DONE;
	}
	strcpy(txTest, "test_CriticalAlarmDueDryerStopButtonPressed");
	switch (iTestState)
	{
		case 0:
			gSimMachine.Commands.xToZero = TRUE;
			nextState();
			break;

		case 1:
			strcpy(txStateDesc, "Waiting the machine to be in Zero");
			TEST_BUSY_CONDITION( gMachine.St.exec.fast < exTimesPreFast + 3 );
			TEST_BUSY_CONDITION( !gMachine.St.Mode.xZero );
			nextState();
			break;

		case 2:
			gSimMachine.Commands.xToAuto = TRUE;
			nextState();
			break;

		case 3:
			strcpy(txStateDesc, "Waiting the machine to be in Auto");
			TEST_BUSY_CONDITION( gLine.Status !=  LINE_IDLE );
			nextState();
			break;

		case 4:
			strcpy(txStateDesc, "Waiting the machine to be ready");
			TEST_BUSY_CONDITION( gMachine.St.exec.fast < exTimesPreFast + 8 );
			gLine.Commands.Print = TRUE;
			nextState();
			break;

		case 5:
			strcpy(txStateDesc, "Waiting the line to start printing");
			TEST_BUSY_CONDITION( gMachine.St.exec.fast < exTimesPreFast + 8 );
			TEST_BUSY_CONDITION( gLine.Status != LINE_PRINTING );
			nextState();
			break;

		case 6:
			strcpy(txStateDesc, "Pressing dryer stop button");
			gDryerAnc.Inputs.xStopButtonPressed=TRUE;
			TEST_BUSY_CONDITION( gLine.Status != LINE_ERROR );
			gDryerAnc.Inputs.xStopButtonPressed=FALSE;
			nextState();
			break;

		case 7:
			strcpy(txStateDesc, "Waiting the line to control stop");
			gMachine.In.Buttons.xReset = TRUE;
			TEST_BUSY_CONDITION( gMachine.St.exec.fast < exTimesPreFast + 8 );
			gSimMachine.Commands.xToZero = TRUE;
			TEST_BUSY_CONDITION( !gMachine.St.Mode.xZero );
			gSimMachine.Commands.xToAuto = TRUE;
			gMachine.In.Buttons.xReset = TRUE;
			nextState();
			break;

		case 8:
			strcpy(txStateDesc, "Waiting the line to be stopped");
			TEST_BUSY_CONDITION( gMachine.St.exec.fast < exTimesPreFast + 8 );
			TEST_BUSY_CONDITION( gLine.Status != LINE_IDLE );
			TEST_ASSERT(gLine.Status == LINE_IDLE);

			iTestState = 0;
			TEST_DONE;

			break;

		default:
			break;
	}
}

_TEST test_CriticalAlarmDueToStackerErrorWhilePrintingLine(void)
{
	if (!gMachine.Pt.xControlledByLine ){
		iTestState = 0;
		TEST_DONE;
	}
	strcpy(txTest, "test_CriticalAlarmDueToStackerErrorWhilePrintingLine");
	switch (iTestState)
	{
		case 0:
			gSimMachine.Commands.xToZero = TRUE;
			nextState();
			break;

		case 1:
			strcpy(txStateDesc, "Waiting the machine to be in Zero");
			TEST_BUSY_CONDITION( gMachine.St.exec.fast < exTimesPreFast + 3 );
			TEST_BUSY_CONDITION( !gMachine.St.Mode.xZero );
			nextState();
			break;

		case 2:
			gSimMachine.Commands.xToAuto = TRUE;
			nextState();
			break;

		case 3:
			strcpy(txStateDesc, "Waiting the machine to be in Auto");
			TEST_BUSY_CONDITION( gLine.Status !=  LINE_IDLE );
			nextState();
			break;

		case 4:
			strcpy(txStateDesc, "Waiting the machine to be ready");
			TEST_BUSY_CONDITION( gMachine.St.exec.fast < exTimesPreFast + 8 );
			gLine.Commands.Print = TRUE;
			nextState();
			break;

		case 5:
			strcpy(txStateDesc, "Waiting the line to start printing");
			TEST_BUSY_CONDITION( gMachine.St.exec.fast < exTimesPreFast + 8 );
			TEST_BUSY_CONDITION( gLine.Status != LINE_PRINTING );
			nextState();
			break;

		case 6:
			strcpy(txStateDesc, "Waiting the line to stop");
			gSimStacker.Commands.CreateError = TRUE;
			TEST_BUSY_CONDITION( gLine.Status != LINE_ERROR );
			gSimStacker.Commands.CreateError = FALSE;
			nextState();
			break;

		case 7:
			strcpy(txStateDesc, "Waiting the line to control stop");
			gMachine.In.Buttons.xReset = TRUE;
			TEST_BUSY_CONDITION( gMachine.St.exec.fast < exTimesPreFast + 8 );
			gSimMachine.Commands.xToZero = TRUE;
			TEST_BUSY_CONDITION( !gMachine.St.Mode.xZero );
			gSimMachine.Commands.xToAuto = TRUE;
			gMachine.In.Buttons.xReset = TRUE;
			nextState();
			break;

		case 8:
			strcpy(txStateDesc, "Waiting the line to be stopped");
			TEST_BUSY_CONDITION( gMachine.St.exec.fast < exTimesPreFast + 8 );
			TEST_BUSY_CONDITION( gLine.Status != LINE_IDLE );
			TEST_ASSERT(gLine.Status == LINE_IDLE);

			iTestState = 0;
			TEST_DONE;

			break;

		default:
			break;
	}
}

_TEST test_CriticalAlarmDueToStackerStopsBeltsWhilePrintingLine(void)
{
	if (!gMachine.Pt.xControlledByLine ){
		iTestState = 0;
		TEST_DONE;
	}
	strcpy(txTest, "test_CriticalAlarmDueToStackerStopsBeltsWhilePrintingLine");
	switch (iTestState)
	{
		case 0:
			gSimMachine.Commands.xToZero = TRUE;
			nextState();
			break;

		case 1:
			strcpy(txStateDesc, "Waiting the machine to be in Zero");
			TEST_BUSY_CONDITION( gMachine.St.exec.fast < exTimesPreFast + 3 );
			TEST_BUSY_CONDITION( !gMachine.St.Mode.xZero );
			nextState();
			break;

		case 2:
			gSimMachine.Commands.xToAuto = TRUE;
			nextState();
			break;

		case 3:
			strcpy(txStateDesc, "Waiting the machine to be in Auto");
			TEST_BUSY_CONDITION( gLine.Status !=  LINE_IDLE );
			nextState();
			break;

		case 4:
			strcpy(txStateDesc, "Waiting the machine to be ready");
			TEST_BUSY_CONDITION( gMachine.St.exec.fast < exTimesPreFast + 8 );
			gLine.Commands.Print = TRUE;
			nextState();
			break;

		case 5:
			strcpy(txStateDesc, "Waiting the line to start printing");
			TEST_BUSY_CONDITION( gMachine.St.exec.fast < exTimesPreFast + 8 );
			TEST_BUSY_CONDITION( gLine.Status != LINE_PRINTING );
			nextState();
			break;

		case 6:
			strcpy(txStateDesc, "Waiting the line to stop");
			gSimStacker.Commands.StopBelts = TRUE;
			TEST_BUSY_CONDITION( gLine.Status != LINE_ERROR );
			gSimStacker.Commands.StopBelts = FALSE;
			nextState();
			break;

		case 7:
			strcpy(txStateDesc, "Waiting the line to control stop");
			gMachine.In.Buttons.xReset = TRUE;
			TEST_BUSY_CONDITION( gMachine.St.exec.fast < exTimesPreFast + 8 );
			gSimMachine.Commands.xToZero = TRUE;
			TEST_BUSY_CONDITION( !gMachine.St.Mode.xZero );
			gSimMachine.Commands.xToAuto = TRUE;
			gMachine.In.Buttons.xReset = TRUE;
			nextState();
			break;

		case 8:
			strcpy(txStateDesc, "Waiting the line to be stopped");
			TEST_BUSY_CONDITION( gMachine.St.exec.fast < exTimesPreFast + 8 );
			TEST_BUSY_CONDITION( gLine.Status != LINE_IDLE );
			TEST_ASSERT(gLine.Status == LINE_IDLE);

			iTestState = 0;
			TEST_DONE;

			break;

		default:
			break;
	}
}

_TEST test_CriticalAlarmDueToOpvErrorWhilePrintingLine(void)
{
	if (!gMachine.St.HwData.xIsWater)
	{
		TEST_DONE;
	}
	if (!gMachine.Pt.xControlledByLine ){
		iTestState = 0;
		TEST_DONE;
	}
	strcpy(txTest, "test_CriticalAlarmDueToOpvErrorWhilePrintingLine");
	switch (iTestState)
	{
		case 0:
			gSimMachine.Commands.xToZero = TRUE;
			nextState();
			break;

		case 1:
			strcpy(txStateDesc, "Waiting the machine to be in Zero");
			TEST_BUSY_CONDITION( gMachine.St.exec.fast < exTimesPreFast + 3 );
			TEST_BUSY_CONDITION( !gMachine.St.Mode.xZero );
			nextState();
			break;

		case 2:
			gSimMachine.Commands.xToAuto = TRUE;
			nextState();
			break;

		case 3:
			strcpy(txStateDesc, "Waiting the machine to be in Auto");
			TEST_BUSY_CONDITION( gLine.Status !=  LINE_IDLE );
			nextState();
			break;

		case 4:
			strcpy(txStateDesc, "Waiting the machine to be ready");
			TEST_BUSY_CONDITION( gMachine.St.exec.fast < exTimesPreFast + 8 );
			gLine.Commands.Print = TRUE;
			nextState();
			break;

		case 5:
			strcpy(txStateDesc, "Waiting the line to start printing");
			TEST_BUSY_CONDITION( gMachine.St.exec.fast < exTimesPreFast + 8 );
			TEST_BUSY_CONDITION( gLine.Status != LINE_PRINTING );
			nextState();
			break;

		case 6:
			strcpy(txStateDesc, "Waiting the line to stop");
			gSimOverVarnish.Commands.CreateError = TRUE;
			TEST_BUSY_CONDITION( gLine.Status != LINE_ERROR );
			gSimOverVarnish.Commands.CreateError = FALSE;
			nextState();
			break;

		case 7:
			strcpy(txStateDesc, "Waiting the line to control stop");
			gMachine.In.Buttons.xReset = TRUE;
			TEST_BUSY_CONDITION( gMachine.St.exec.fast < exTimesPreFast + 8 );
			gSimMachine.Commands.xToZero = TRUE;
			TEST_BUSY_CONDITION( !gMachine.St.Mode.xZero );
			gSimMachine.Commands.xToAuto = TRUE;
			gMachine.In.Buttons.xReset = TRUE;
			nextState();
			break;

		case 8:
			strcpy(txStateDesc, "Waiting the line to be stopped");
			TEST_BUSY_CONDITION( gMachine.St.exec.fast < exTimesPreFast + 8 );
			TEST_BUSY_CONDITION( gLine.Status != LINE_IDLE );
			TEST_ASSERT(gLine.Status == LINE_IDLE);

			iTestState = 0;
			TEST_DONE;

			break;

		default:
			break;
	}
}

_TEST test_OutOfAutoWhilePrintingLine(void)
{
	if (!gMachine.Pt.xControlledByLine ){
		iTestState = 0;
		TEST_DONE;
	}
	strcpy(txTest, "test_OutOfAutoWhilePrintingLine");
	switch (iTestState)
	{
		case 0:
			gSimMachine.Commands.xToZero = TRUE;
			nextState();
			break;

		case 1:
			strcpy(txStateDesc, "Waiting the machine to be in Zero");
			TEST_BUSY_CONDITION( gMachine.St.exec.fast < exTimesPreFast + 3 );
			TEST_BUSY_CONDITION( !gMachine.St.Mode.xZero );
			nextState();
			break;

		case 2:
			gSimMachine.Commands.xToAuto = TRUE;
			nextState();
			break;

		case 3:
			strcpy(txStateDesc, "Waiting the machine to be in Auto");
			TEST_BUSY_CONDITION( !gMachine.St.Mode.xAuto );
			gMachine.In.Buttons.xReset = TRUE;
			nextState();
			break;

		case 4:
			strcpy(txStateDesc, "Waiting the machine to be ready");
			TEST_BUSY_CONDITION( gMachine.St.exec.fast < exTimesPreFast + 8 );
			gLine.Commands.Print = TRUE;
			nextState();
			break;

		case 5:
			strcpy(txStateDesc, "Waiting the line to start printing");
			TEST_BUSY_CONDITION( gMachine.St.exec.fast < exTimesPreFast + 8 );
			TEST_BUSY_CONDITION( gLine.Status != LINE_PRINTING );
			nextState();
			break;

		case 6:
			strcpy(txStateDesc, "Waiting the line to be in error state");
			gSimMachine.Commands.xToAuto = FALSE;
			gSimMachine.Commands.xToZero = TRUE;
			TEST_BUSY_CONDITION( gLine.Status != LINE_STOPPED );
			nextState();
			break;

		case 7:
			strcpy(txStateDesc, "Waiting the line to be stopped");
			TEST_BUSY_CONDITION( gMachine.St.exec.fast < exTimesPreFast + 8 );
			TEST_ASSERT(gLine.Status == LINE_STOPPED);

			iTestState = 0;
			TEST_DONE;

			break;

		default:
			break;
	}
}

_TEST test_BarsComeBackToCapAfterZeroModeWhilePrintingLine(void)
{
	if (!gMachine.Pt.xControlledByLine ){
		iTestState = 0;
		TEST_DONE;
	}
	strcpy(txTest, "test_BarsComeBackToCapAfterZeroModeWhilePrintingLine");
	switch (iTestState)
	{
		case 0:
			gSimMachine.Commands.xToZero = TRUE;
			nextState();
			break;

		case 1:
			strcpy(txStateDesc, "Waiting the machine to be in Zero");
			TEST_BUSY_CONDITION( gMachine.St.exec.fast < exTimesPreFast + 3 );
			TEST_BUSY_CONDITION( !gMachine.St.Mode.xZero );
			nextState();
			break;

		case 2:
			gSimMachine.Commands.xToAuto = TRUE;
			nextState();
			break;

		case 3:
			strcpy(txStateDesc, "Waiting the machine to be in Auto");
			TEST_BUSY_CONDITION( !gMachine.St.Mode.xAuto );
			gMachine.In.Buttons.xReset = TRUE;
			nextState();
			break;

		case 4:
			strcpy(txStateDesc, "Waiting the machine to be ready");
			TEST_BUSY_CONDITION( gMachine.St.exec.fast < exTimesPreFast + 8 );
			gLine.Commands.Print = TRUE;
			nextState();
			break;

		case 5:
			strcpy(txStateDesc, "Waiting the line to start printing");
			TEST_BUSY_CONDITION( gMachine.St.exec.fast < exTimesPreFast + 8 );
			TEST_BUSY_CONDITION( gLine.Status != LINE_PRINTING );
			nextState();
			break;

		case 6:
			strcpy(txStateDesc, "Waiting the line to be in error state");
			gSimMachine.Commands.xToZero = TRUE;
			nextState();
			break;

		case 7:
			strcpy(txStateDesc, "Waiting the line to be stopped");
			TEST_BUSY_CONDITION( gMachine.St.exec.fast < exTimesPreFast + 8 );
			TEST_BUSY_CONDITION( gLine.Status != LINE_STOPPED );
			nextState();
			break;

		case 8:
			strcpy(txStateDesc, "Setting automatic mode");
			TEST_BUSY_CONDITION( gMachine.St.exec.fast < exTimesPreFast + 8 );
			gSimMachine.Commands.xToAuto = TRUE;
			TEST_BUSY_CONDITION( !gMachine.St.Mode.xAuto );
			gMachine.In.Buttons.xReset = TRUE;
			nextState();
			break;
```
